LIN {X 0,Y 190.257,Z 771.261,A -85,B 0,C 180,E1 -26791.509,E2 -26791.509} C_VEL
LIN {X 0,Y 190.301,Z 771.078,A -85,B 0,C 180,E1 -26791.798,E2 -26791.798} C_VEL
LIN {X 0,Y 189.39,Z 772.436,A -85,B 0,C 180,E1 -26792.401,E2 -26792.401} C_VEL
LIN {X 0,Y 186.858,Z 776.269,A -85,B 0,C 180,E1 -26793.185,E2 -26793.185} C_VEL
LIN {X 0,Y 179.691,Z 786.165,A -85,B 0,C 180,E1 -26794.58,E2 -26794.58} C_VEL
LIN {X 0,Y 172.891,Z 794.099,A -85,B 0,C 180,E1 -26795.858,E2 -26795.858} C_VEL
LIN {X 0,Y 164.978,Z 801.951,A -85,B 0,C 180,E1 -26797.455,E2 -26797.455} C_VEL
LIN {X 0,Y 154.213,Z 810.811,A -85,B 0,C 180,E1 -26800.013,E2 -26800.013} C_VEL
LIN {X 0,Y 146.324,Z 816.184,A -85,B 0,C 180,E1 -26802.169,E2 -26802.169} C_VEL
LIN {X 0,Y 137.196,Z 821.36,A -85,B 0,C 180,E1 -26805.159,E2 -26805.159} C_VEL
LIN {X 0,Y 129.179,Z 825.032,A -85,B 0,C 180,E1 -26808.3,E2 -26808.3} C_VEL
LIN {X 0,Y 120.494,Z 828.105,A -85,B 0,C 180,E1 -26812.517,E2 -26812.517} C_VEL
LIN {X 0,Y 112.556,Z 829.932,A -85,B 0,C 180,E1 -26817.398,E2 -26817.398} C_VEL
LIN {X 0,Y 104.804,Z 830.561,A -85,B 0,C 180,E1 -26823.845,E2 -26823.845} C_VEL
LIN {X 0,Y 99.766,Z 830.01,A -85,B 0,C 180,E1 -26829.549,E2 -26829.549} C_VEL
LIN {X 0,Y 95.081,Z 828.076,A -85,B 0,C 180,E1 -26837.197,E2 -26837.197} C_VEL
LIN {X 0,Y 92.422,Z 825.28,A -85,B 0,C 180,E1 -26844.158,E2 -26844.158} C_VEL
LIN {X 0,Y 91.047,Z 820.547,A -85,B 0,C 180,E1 -26852.706,E2 -26852.706} C_VEL
LIN {X 0,Y 91.19,Z 815.515,A -85,B 0,C 180,E1 -26859.592,E2 -26859.592} C_VEL
LIN {X 0,Y 91.968,Z 810.446,A -85,B 0,C 180,E1 -26865.175,E2 -26865.175} C_VEL
LIN {X 0,Y 93.476,Z 803.521,A -85,B 0,C 180,E1 -26871.266,E2 -26871.266} C_VEL
LIN {X 0,Y 95.726,Z 795.077,A -85,B 0,C 180,E1 -26877.134,E2 -26877.134} C_VEL
LIN {X 0,Y 98.846,Z 784.708,A -85,B 0,C 180,E1 -26882.716,E2 -26882.716} C_VEL
LIN {X 0,Y 102.013,Z 773.87,A -85,B 0,C 180,E1 -26887.138,E2 -26887.138} C_VEL
LIN {X 0,Y 105.077,Z 762.843,A -85,B 0,C 180,E1 -26890.585,E2 -26890.585} C_VEL
LIN {X 0,Y 107.937,Z 750.627,A -85,B 0,C 180,E1 -26893.49,E2 -26893.49} C_VEL
LIN {X 0,Y 110.363,Z 737.817,A -85,B 0,C 180,E1 -26895.696,E2 -26895.696} C_VEL
LIN {X 0,Y 112.229,Z 724.1,A -85,B 0,C 180,E1 -26897.338,E2 -26897.338} C_VEL
LIN {X 0,Y 116.253,Z 682.181,A -85,B 0,C 180,E1 -26900.432,E2 -26900.432} C_VEL
LIN {X 0,Y 115.274,Z 679.01,A -85,B 0,C 180,E1 -26901.012,E2 -26901.012} C_VEL
LIN {X 0,Y 108.762,Z 662.742,A -85,B 0,C 180,E1 -26904.591,E2 -26904.591} C_VEL
LIN {X 0,Y 103.474,Z 650.911,A -85,B 0,C 180,E1 -26907.786,E2 -26907.786} C_VEL
LIN {X 0,Y 97.006,Z 638.252,A -85,B 0,C 180,E1 -26912.011,E2 -26912.011} C_VEL
LIN {X 0,Y 95.064,Z 635.94,A -85,B 0,C 180,E1 -26913.23,E2 -26913.23} C_VEL
LIN {X 0,Y 94.335,Z 633.735,A -85,B 0,C 180,E1 -26914.036,E2 -26914.036} C_VEL
LIN {X 0,Y 94.213,Z 633.749,A -85,B 0,C 180,E1 -26918.585,E2 -26918.585} C_VEL
LIN {X 0,Y 94.049,Z 633.77,A -85,B 0,C 180,E1 -26923.726,E2 -26923.726} C_VEL
LIN {X 0,Y 93.696,Z 633.798,A -85,B 0,C 180,E1 -26932.032,E2 -26932.032} C_VEL
LIN {X 0,Y 93.625,Z 633.822,A -85,B 0,C 180,E1 -26936.774,E2 -26936.774} C_VEL
LIN {X 0,Y 93.591,Z 633.786,A -85,B 0,C 180,E1 -26944.309,E2 -26944.309} C_VEL
LIN {X 0,Y 93.537,Z 633.831,A -85,B 0,C 180,E1 -26952.555,E2 -26952.555} C_VEL
LIN {X 0,Y 93.542,Z 633.801,A -85,B 0,C 180,E1 -26958.711,E2 -26958.711} C_VEL
LIN {X 0,Y 93.596,Z 633.788,A -85,B 0,C 180,E1 -26965.695,E2 -26965.695} C_VEL
LIN {X 0,Y 93.675,Z 633.815,A -85,B 0,C 180,E1 -26974.208,E2 -26974.208} C_VEL
LIN {X 0,Y 93.696,Z 633.798,A -85,B 0,C 180,E1 -26977.974,E2 -26977.974} C_VEL
LIN {X 0,Y 94.075,Z 633.734,A -85,B 0,C 180,E1 -26987.05,E2 -26987.05} C_VEL
LIN {X 0,Y 94.184,Z 633.749,A -85,B 0,C 180,E1 -26991.418,E2 -26991.418} C_VEL
LIN {X 0,Y 94.782,Z 633.646,A -85,B 0,C 180,E1 -27000.001,E2 -27000.001} C_VEL
LIN {X 0,Y 94.172,Z 633.755,A -85,B 0,C 180,E1 -27008.585,E2 -27008.585} C_VEL
LIN {X 0,Y 93.971,Z 633.763,A -85,B 0,C 180,E1 -27013.51,E2 -27013.51} C_VEL
LIN {X 0,Y 93.693,Z 633.817,A -85,B 0,C 180,E1 -27022.028,E2 -27022.028} C_VEL
LIN {X 0,Y 93.627,Z 633.827,A -85,B 0,C 180,E1 -27029.204,E2 -27029.204} C_VEL
LIN {X 0,Y 93.635,Z 633.826,A -85,B 0,C 180,E1 -27029.51,E2 -27029.51} C_VEL
LIN {X 0,Y 94.623,Z 636.565,A -85,B 0,C 180,E1 -27030.398,E2 -27030.398} C_VEL
LIN {X 0,Y 96.199,Z 638.846,A -85,B 0,C 180,E1 -27031.453,E2 -27031.453} C_VEL
LIN {X 0,Y 103.193,Z 651.438,A -85,B 0,C 180,E1 -27035.955,E2 -27035.955} C_VEL
LIN {X 0,Y 108.688,Z 666.292,A -85,B 0,C 180,E1 -27039.528,E2 -27039.528} C_VEL
LIN {X 0,Y 114.31,Z 684.536,A -85,B 0,C 180,E1 -27043.054,E2 -27043.054} C_VEL
LIN {X 0,Y 115.161,Z 702.412,A -85,B 0,C 180,E1 -27045.026,E2 -27045.026} C_VEL
LIN {X 0,Y 111.773,Z 738.131,A -85,B 0,C 180,E1 -27047.773,E2 -27047.773} C_VEL
LIN {X 0,Y 109.635,Z 752.163,A -85,B 0,C 180,E1 -27049.525,E2 -27049.525} C_VEL
LIN {X 0,Y 107.125,Z 764.111,A -85,B 0,C 180,E1 -27051.681,E2 -27051.681} C_VEL
LIN {X 0,Y 103.733,Z 777.276,A -85,B 0,C 180,E1 -27054.978,E2 -27054.978} C_VEL
LIN {X 0,Y 100.451,Z 788.747,A -85,B 0,C 180,E1 -27058.932,E2 -27058.932} C_VEL
LIN {X 0,Y 97.658,Z 798.326,A -85,B 0,C 180,E1 -27063.265,E2 -27063.265} C_VEL
LIN {X 0,Y 95.188,Z 807.085,A -85,B 0,C 180,E1 -27068.331,E2 -27068.331} C_VEL
LIN {X 0,Y 93.458,Z 814.321,A -85,B 0,C 180,E1 -27073.616,E2 -27073.616} C_VEL
LIN {X 0,Y 92.315,Z 821.391,A -85,B 0,C 180,E1 -27080.132,E2 -27080.132} C_VEL
LIN {X 0,Y 92.185,Z 826.13,A -85,B 0,C 180,E1 -27085.623,E2 -27085.623} C_VEL
LIN {X 0,Y 92.19,Z 829.203,A -85,B 0,C 180,E1 -27089.995,E2 -27089.995} C_VEL
LIN {X 0,Y 91.921,Z 832.559,A -85,B 0,C 180,E1 -27096.306,E2 -27096.306} C_VEL
LIN {X 0,Y 92.284,Z 835.092,A -85,B 0,C 180,E1 -27103.202,E2 -27103.202} C_VEL
LIN {X 0,Y 94.653,Z 837.065,A -85,B 0,C 180,E1 -27111.788,E2 -27111.788} C_VEL
LIN {X 0,Y 99.342,Z 837.643,A -85,B 0,C 180,E1 -27119.679,E2 -27119.679} C_VEL
LIN {X 0,Y 105.831,Z 836.874,A -85,B 0,C 180,E1 -27126.698,E2 -27126.698} C_VEL
LIN {X 0,Y 113.876,Z 834.76,A -85,B 0,C 180,E1 -27132.751,E2 -27132.751} C_VEL
LIN {X 0,Y 123.232,Z 831.198,A -85,B 0,C 180,E1 -27137.845,E2 -27137.845} C_VEL
LIN {X 0,Y 133.648,Z 826.087,A -85,B 0,C 180,E1 -27142.067,E2 -27142.067} C_VEL
LIN {X 0,Y 142.003,Z 821.149,A -85,B 0,C 180,E1 -27144.742,E2 -27144.742} C_VEL
LIN {X 0,Y 152.185,Z 813.997,A -85,B 0,C 180,E1 -27147.431,E2 -27147.431} C_VEL
LIN {X 0,Y 161.26,Z 806.403,A -85,B 0,C 180,E1 -27149.394,E2 -27149.394} C_VEL
LIN {X 0,Y 170.664,Z 797.142,A -85,B 0,C 180,E1 -27151.049,E2 -27151.049} C_VEL
LIN {X 0,Y 179.448,Z 786.784,A -85,B 0,C 180,E1 -27152.381,E2 -27152.381} C_VEL
LIN {X 0,Y 184.99,Z 779.053,A -85,B 0,C 180,E1 -27153.104,E2 -27153.104} C_VEL
LIN {X 0,Y 185.21,Z 778.645,A -85,B 0,C 180,E1 -27153.656,E2 -27153.656} C_VEL
LIN {X 0,Y 177.086,Z 789.352,A -85,B 0,C 180,E1 -27155.058,E2 -27155.058} C_VEL
LIN {X 0,Y 172.891,Z 794.099,A -85,B 0,C 180,E1 -27155.858,E2 -27155.858} C_VEL
LIN {X 0,Y 168.899,Z 798.22,A -85,B 0,C 180,E1 -27156.407,E2 -27156.407} C_VEL
LIN {X 0,Y 161.572,Z 804.876,A -85,B 0,C 180,E1 -27156.817,E2 -27156.817} C_VEL
LIN {X 0,Y 153.89,Z 810.838,A -85,B 0,C 180,E1 -27157.356,E2 -27157.356} C_VEL
LIN {X 0,Y 149.397,Z 813.899,A -85,B 0,C 180,E1 -27158.148,E2 -27158.148} C_VEL
LIN {X 0,Y 139.254,Z 819.917,A -85,B 0,C 180,E1 -27160.848,E2 -27160.848} C_VEL
LIN {X 0,Y 129.108,Z 824.664,A -85,B 0,C 180,E1 -27164.206,E2 -27164.206} C_VEL
LIN {X 0,Y 122.663,Z 827.054,A -85,B 0,C 180,E1 -27166.751,E2 -27166.751} C_VEL
LIN {X 0,Y 113.839,Z 829.524,A -85,B 0,C 180,E1 -27171.006,E2 -27171.006} C_VEL
LIN {X 0,Y 105.533,Z 830.874,A -85,B 0,C 180,E1 -27176.181,E2 -27176.181} C_VEL
LIN {X 0,Y 98.447,Z 831.013,A -85,B 0,C 180,E1 -27182.063,E2 -27182.063} C_VEL
LIN {X 0,Y 92.478,Z 829.966,A -85,B 0,C 180,E1 -27188.933,E2 -27188.933} C_VEL
LIN {X 0,Y 87.974,Z 827.723,A -85,B 0,C 180,E1 -27196.554,E2 -27196.554} C_VEL
LIN {X 0,Y 85.101,Z 824.276,A -85,B 0,C 180,E1 -27204.725,E2 -27204.725} C_VEL
LIN {X 0,Y 83.943,Z 819.532,A -85,B 0,C 180,E1 -27213.161,E2 -27213.161} C_VEL
LIN {X 0,Y 84.158,Z 814.597,A -85,B 0,C 180,E1 -27220.015,E2 -27220.015} C_VEL
LIN {X 0,Y 85.397,Z 807.511,A -85,B 0,C 180,E1 -27227.789,E2 -27227.789} C_VEL
LIN {X 0,Y 87.491,Z 799.088,A -85,B 0,C 180,E1 -27234.89,E2 -27234.89} C_VEL
LIN {X 0,Y 90.326,Z 789.576,A -85,B 0,C 180,E1 -27241.072,E2 -27241.072} C_VEL
LIN {X 0,Y 93.463,Z 779.613,A -85,B 0,C 180,E1 -27245.988,E2 -27245.988} C_VEL
LIN {X 0,Y 96.948,Z 767.721,A -85,B 0,C 180,E1 -27250.458,E2 -27250.458} C_VEL
LIN {X 0,Y 99.998,Z 756.271,A -85,B 0,C 180,E1 -27253.677,E2 -27253.677} C_VEL
LIN {X 0,Y 102.829,Z 743.465,A -85,B 0,C 180,E1 -27256.32,E2 -27256.32} C_VEL
LIN {X 0,Y 105.103,Z 729.84,A -85,B 0,C 180,E1 -27258.31,E2 -27258.31} C_VEL
LIN {X 0,Y 107.076,Z 711.899,A -85,B 0,C 180,E1 -27259.909,E2 -27259.909} C_VEL
LIN {X 0,Y 109.842,Z 683.218,A -85,B 0,C 180,E1 -27262.095,E2 -27262.095} C_VEL
LIN {X 0,Y 103.379,Z 666.533,A -85,B 0,C 180,E1 -27266.022,E2 -27266.022} C_VEL
LIN {X 0,Y 98.287,Z 654.89,A -85,B 0,C 180,E1 -27269.36,E2 -27269.36} C_VEL
LIN {X 0,Y 92.53,Z 643.401,A -85,B 0,C 180,E1 -27273.467,E2 -27273.467} C_VEL
LIN {X 0,Y 90.263,Z 640.187,A -85,B 0,C 180,E1 -27275.111,E2 -27275.111} C_VEL
LIN {X 0,Y 89.464,Z 638.976,A -85,B 0,C 180,E1 -27275.726,E2 -27275.726} C_VEL
LIN {X 0,Y 87.736,Z 636.65,A -85,B 0,C 180,E1 -27277.051,E2 -27277.051} C_VEL
LIN {X 0,Y 87.154,Z 634.627,A -85,B 0,C 180,E1 -27277.826,E2 -27277.826} C_VEL
LIN {X 0,Y 86.952,Z 634.654,A -85,B 0,C 180,E1 -27284.092,E2 -27284.092} C_VEL
LIN {X 0,Y 86.59,Z 634.695,A -85,B 0,C 180,E1 -27293.948,E2 -27293.948} C_VEL
LIN {X 0,Y 86.478,Z 634.702,A -85,B 0,C 180,E1 -27299.189,E2 -27299.189} C_VEL
LIN {X 0,Y 86.51,Z 634.671,A -85,B 0,C 180,E1 -27305.67,E2 -27305.67} C_VEL
LIN {X 0,Y 86.481,Z 634.71,A -85,B 0,C 180,E1 -27312.997,E2 -27312.997} C_VEL
LIN {X 0,Y 86.464,Z 634.672,A -85,B 0,C 180,E1 -27319.44,E2 -27319.44} C_VEL
LIN {X 0,Y 86.54,Z 634.661,A -85,B 0,C 180,E1 -27325.357,E2 -27325.357} C_VEL
LIN {X 0,Y 86.59,Z 634.699,A -85,B 0,C 180,E1 -27333.238,E2 -27333.238} C_VEL
LIN {X 0,Y 86.638,Z 634.648,A -85,B 0,C 180,E1 -27341.067,E2 -27341.067} C_VEL
LIN {X 0,Y 86.938,Z 634.611,A -85,B 0,C 180,E1 -27345.965,E2 -27345.965} C_VEL
LIN {X 0,Y 87.093,Z 634.629,A -85,B 0,C 180,E1 -27350.713,E2 -27350.713} C_VEL
LIN {X 0,Y 87.712,Z 634.525,A -85,B 0,C 180,E1 -27360.001,E2 -27360.001} C_VEL
LIN {X 0,Y 87.074,Z 634.639,A -85,B 0,C 180,E1 -27369.29,E2 -27369.29} C_VEL
LIN {X 0,Y 86.868,Z 634.644,A -85,B 0,C 180,E1 -27374.047,E2 -27374.047} C_VEL
LIN {X 0,Y 86.627,Z 634.693,A -85,B 0,C 180,E1 -27378.937,E2 -27378.937} C_VEL
LIN {X 0,Y 86.629,Z 634.683,A -85,B 0,C 180,E1 -27385.699,E2 -27385.699} C_VEL
LIN {X 0,Y 87.657,Z 637.659,A -85,B 0,C 180,E1 -27386.827,E2 -27386.827} C_VEL
LIN {X 0,Y 89.274,Z 639.751,A -85,B 0,C 180,E1 -27388.058,E2 -27388.058} C_VEL
LIN {X 0,Y 95.254,Z 650.213,A -85,B 0,C 180,E1 -27392.495,E2 -27392.495} C_VEL
LIN {X 0,Y 98.46,Z 656.546,A -85,B 0,C 180,E1 -27394.668,E2 -27394.668} C_VEL
LIN {X 0,Y 104.026,Z 672.659,A -85,B 0,C 180,E1 -27398.678,E2 -27398.678} C_VEL
LIN {X 0,Y 108.21,Z 687.138,A -85,B 0,C 180,E1 -27401.583,E2 -27401.583} C_VEL
LIN {X 0,Y 108.806,Z 702.893,A -85,B 0,C 180,E1 -27403.389,E2 -27403.389} C_VEL
LIN {X 0,Y 105.359,Z 737.654,A -85,B 0,C 180,E1 -27406.201,E2 -27406.201} C_VEL
LIN {X 0,Y 103.128,Z 751.621,A -85,B 0,C 180,E1 -27408.028,E2 -27408.028} C_VEL
LIN {X 0,Y 100.378,Z 764.08,A -85,B 0,C 180,E1 -27410.41,E2 -27410.41} C_VEL
LIN {X 0,Y 97.072,Z 776.396,A -85,B 0,C 180,E1 -27413.681,E2 -27413.681} C_VEL
LIN {X 0,Y 93.764,Z 787.607,A -85,B 0,C 180,E1 -27417.715,E2 -27417.715} C_VEL
LIN {X 0,Y 90.803,Z 797.289,A -85,B 0,C 180,E1 -27422.324,E2 -27422.324} C_VEL
LIN {X 0,Y 88.22,Z 806.145,A -85,B 0,C 180,E1 -27427.76,E2 -27427.76} C_VEL
LIN {X 0,Y 86.147,Z 814.79,A -85,B 0,C 180,E1 -27434.62,E2 -27434.62} C_VEL
LIN {X 0,Y 85.214,Z 821.7,A -85,B 0,C 180,E1 -27441.773,E2 -27441.773} C_VEL
LIN {X 0,Y 85.191,Z 826.219,A -85,B 0,C 180,E1 -27447.631,E2 -27447.631} C_VEL
LIN {X 0,Y 85.153,Z 829.094,A -85,B 0,C 180,E1 -27452.36,E2 -27452.36} C_VEL
LIN {X 0,Y 84.943,Z 832.374,A -85,B 0,C 180,E1 -27459.52,E2 -27459.52} C_VEL
LIN {X 0,Y 86.475,Z 835.317,A -85,B 0,C 180,E1 -27468.965,E2 -27468.965} C_VEL
LIN {X 0,Y 90.35,Z 836.847,A -85,B 0,C 180,E1 -27477.816,E2 -27477.816} C_VEL
LIN {X 0,Y 96.496,Z 837.06,A -85,B 0,C 180,E1 -27485.632,E2 -27485.632} C_VEL
LIN {X 0,Y 104.304,Z 835.891,A -85,B 0,C 180,E1 -27492.355,E2 -27492.355} C_VEL
LIN {X 0,Y 113.522,Z 833.378,A -85,B 0,C 180,E1 -27497.973,E2 -27497.973} C_VEL
LIN {X 0,Y 121.231,Z 830.566,A -85,B 0,C 180,E1 -27501.495,E2 -27501.495} C_VEL
LIN {X 0,Y 132.291,Z 825.471,A -85,B 0,C 180,E1 -27505.424,E2 -27505.424} C_VEL
LIN {X 0,Y 141.025,Z 820.498,A -85,B 0,C 180,E1 -27507.902,E2 -27507.902} C_VEL
LIN {X 0,Y 151.627,Z 813.379,A -85,B 0,C 180,E1 -27510.345,E2 -27510.345} C_VEL
LIN {X 0,Y 161.018,Z 805.796,A -85,B 0,C 180,E1 -27512.105,E2 -27512.105} C_VEL
LIN {X 0,Y 167.484,Z 799.75,A -85,B 0,C 180,E1 -27513.122,E2 -27513.122} C_VEL
LIN {X 0,Y 169.396,Z 797.758,A -85,B 0,C 180,E1 -27513.97,E2 -27513.97} C_VEL
LIN {X 0,Y 160.59,Z 805.702,A -85,B 0,C 180,E1 -27515.652,E2 -27515.652} C_VEL
LIN {X 0,Y 150.031,Z 813.478,A -85,B 0,C 180,E1 -27517.991,E2 -27517.991} C_VEL
LIN {X 0,Y 149.397,Z 813.899,A -85,B 0,C 180,E1 -27518.148,E2 -27518.148} C_VEL
LIN {X 0,Y 144.757,Z 816.802,A -85,B 0,C 180,E1 -27519.036,E2 -27519.036} C_VEL
LIN {X 0,Y 136.239,Z 821.334,A -85,B 0,C 180,E1 -27520.012,E2 -27520.012} C_VEL
LIN {X 0,Y 127.551,Z 825.143,A -85,B 0,C 180,E1 -27521.2,E2 -27521.2} C_VEL
LIN {X 0,Y 122.718,Z 826.849,A -85,B 0,C 180,E1 -27522.485,E2 -27522.485} C_VEL
LIN {X 0,Y 114.479,Z 829.304,A -85,B 0,C 180,E1 -27525.784,E2 -27525.784} C_VEL
LIN {X 0,Y 107.282,Z 830.741,A -85,B 0,C 180,E1 -27529.285,E2 -27529.285} C_VEL
LIN {X 0,Y 98.829,Z 831.572,A -85,B 0,C 180,E1 -27534.558,E2 -27534.558} C_VEL
LIN {X 0,Y 91.366,Z 831.247,A -85,B 0,C 180,E1 -27540.858,E2 -27540.858} C_VEL
LIN {X 0,Y 85.202,Z 829.729,A -85,B 0,C 180,E1 -27548.214,E2 -27548.214} C_VEL
LIN {X 0,Y 80.612,Z 826.993,A -85,B 0,C 180,E1 -27556.482,E2 -27556.482} C_VEL
LIN {X 0,Y 77.813,Z 823.015,A -85,B 0,C 180,E1 -27565.434,E2 -27565.434} C_VEL
LIN {X 0,Y 76.866,Z 817.762,A -85,B 0,C 180,E1 -27574.636,E2 -27574.636} C_VEL
LIN {X 0,Y 77.27,Z 812.753,A -85,B 0,C 180,E1 -27581.579,E2 -27581.579} C_VEL
LIN {X 0,Y 78.524,Z 806.204,A -85,B 0,C 180,E1 -27588.885,E2 -27588.885} C_VEL
LIN {X 0,Y 80.91,Z 797.234,A -85,B 0,C 180,E1 -27596.678,E2 -27596.678} C_VEL
LIN {X 0,Y 84.32,Z 786.507,A -85,B 0,C 180,E1 -27603.637,E2 -27603.637} C_VEL
LIN {X 0,Y 87.783,Z 775.869,A -85,B 0,C 180,E1 -27608.795,E2 -27608.795} C_VEL
LIN {X 0,Y 91.421,Z 763.754,A -85,B 0,C 180,E1 -27613.167,E2 -27613.167} C_VEL
LIN {X 0,Y 94.498,Z 752.043,A -85,B 0,C 180,E1 -27616.297,E2 -27616.297} C_VEL
LIN {X 0,Y 97.388,Z 738.237,A -85,B 0,C 180,E1 -27618.911,E2 -27618.911} C_VEL
LIN {X 0,Y 99.344,Z 725.28,A -85,B 0,C 180,E1 -27620.602,E2 -27620.602} C_VEL
LIN {X 0,Y 103.501,Z 684.743,A -85,B 0,C 180,E1 -27623.911,E2 -27623.911} C_VEL
LIN {X 0,Y 97.838,Z 669.858,A -85,B 0,C 180,E1 -27627.699,E2 -27627.699} C_VEL
LIN {X 0,Y 93.131,Z 658.831,A -85,B 0,C 180,E1 -27631.087,E2 -27631.087} C_VEL
LIN {X 0,Y 87.987,Z 648.291,A -85,B 0,C 180,E1 -27635.173,E2 -27635.173} C_VEL
LIN {X 0,Y 84.861,Z 643.815,A -85,B 0,C 180,E1 -27637.652,E2 -27637.652} C_VEL
LIN {X 0,Y 82.422,Z 639.977,A -85,B 0,C 180,E1 -27639.824,E2 -27639.824} C_VEL
LIN {X 0,Y 80.655,Z 637.846,A -85,B 0,C 180,E1 -27641.419,E2 -27641.419} C_VEL
LIN {X 0,Y 79.921,Z 635.526,A -85,B 0,C 180,E1 -27642.481,E2 -27642.481} C_VEL
LIN {X 0,Y 79.516,Z 635.555,A -85,B 0,C 180,E1 -27650.71,E2 -27650.71} C_VEL
LIN {X 0,Y 79.485,Z 635.58,A -85,B 0,C 180,E1 -27657.849,E2 -27657.849} C_VEL
LIN {X 0,Y 79.381,Z 635.559,A -85,B 0,C 180,E1 -27662.094,E2 -27662.094} C_VEL
LIN {X 0,Y 79.369,Z 635.58,A -85,B 0,C 180,E1 -27668.311,E2 -27668.311} C_VEL
LIN {X 0,Y 79.39,Z 635.586,A -85,B 0,C 180,E1 -27675.096,E2 -27675.096} C_VEL
LIN {X 0,Y 79.393,Z 635.536,A -85,B 0,C 180,E1 -27682.824,E2 -27682.824} C_VEL
LIN {X 0,Y 79.385,Z 635.575,A -85,B 0,C 180,E1 -27687.915,E2 -27687.915} C_VEL
LIN {X 0,Y 79.531,Z 635.578,A -85,B 0,C 180,E1 -27693.779,E2 -27693.779} C_VEL
LIN {X 0,Y 79.511,Z 635.549,A -85,B 0,C 180,E1 -27699.296,E2 -27699.296} C_VEL
LIN {X 0,Y 79.832,Z 635.491,A -85,B 0,C 180,E1 -27705.575,E2 -27705.575} C_VEL
LIN {X 0,Y 79.976,Z 635.511,A -85,B 0,C 180,E1 -27709.878,E2 -27709.878} C_VEL
LIN {X 0,Y 80.641,Z 635.404,A -85,B 0,C 180,E1 -27720.001,E2 -27720.001} C_VEL
LIN {X 0,Y 79.951,Z 635.526,A -85,B 0,C 180,E1 -27730.126,E2 -27730.126} C_VEL
LIN {X 0,Y 79.7,Z 635.535,A -85,B 0,C 180,E1 -27735.341,E2 -27735.341} C_VEL
LIN {X 0,Y 79.508,Z 635.586,A -85,B 0,C 180,E1 -27741.046,E2 -27741.046} C_VEL
LIN {X 0,Y 80.462,Z 638.379,A -85,B 0,C 180,E1 -27742.298,E2 -27742.298} C_VEL
LIN {X 0,Y 82.444,Z 640.682,A -85,B 0,C 180,E1 -27744.054,E2 -27744.054} C_VEL
LIN {X 0,Y 84.504,Z 644.136,A -85,B 0,C 180,E1 -27745.936,E2 -27745.936} C_VEL
LIN {X 0,Y 88.954,Z 651.914,A -85,B 0,C 180,E1 -27749.662,E2 -27749.662} C_VEL
LIN {X 0,Y 93.093,Z 659.974,A -85,B 0,C 180,E1 -27752.802,E2 -27752.802} C_VEL
LIN {X 0,Y 98.329,Z 675.548,A -85,B 0,C 180,E1 -27756.93,E2 -27756.93} C_VEL
LIN {X 0,Y 102.085,Z 689.101,A -85,B 0,C 180,E1 -27759.876,E2 -27759.876} C_VEL
LIN {X 0,Y 102.526,Z 703.086,A -85,B 0,C 180,E1 -27761.586,E2 -27761.586} C_VEL
LIN {X 0,Y 98.903,Z 737.844,A -85,B 0,C 180,E1 -27764.551,E2 -27764.551} C_VEL
LIN {X 0,Y 96.715,Z 750.887,A -85,B 0,C 180,E1 -27766.34,E2 -27766.34} C_VEL
LIN {X 0,Y 93.883,Z 763.305,A -85,B 0,C 180,E1 -27768.803,E2 -27768.803} C_VEL
LIN {X 0,Y 90.418,Z 775.691,A -85,B 0,C 180,E1 -27772.252,E2 -27772.252} C_VEL
LIN {X 0,Y 87.128,Z 786.446,A -85,B 0,C 180,E1 -27776.314,E2 -27776.314} C_VEL
LIN {X 0,Y 83.991,Z 796.258,A -85,B 0,C 180,E1 -27781.235,E2 -27781.235} C_VEL
LIN {X 0,Y 81.262,Z 805.169,A -85,B 0,C 180,E1 -27787.09,E2 -27787.09} C_VEL
LIN {X 0,Y 79.113,Z 813.861,A -85,B 0,C 180,E1 -27794.538,E2 -27794.538} C_VEL
LIN {X 0,Y 78.268,Z 819.777,A -85,B 0,C 180,E1 -27801.021,E2 -27801.021} C_VEL
LIN {X 0,Y 78.216,Z 824.532,A -85,B 0,C 180,E1 -27807.419,E2 -27807.419} C_VEL
LIN {X 0,Y 78.216,Z 827.636,A -85,B 0,C 180,E1 -27812.569,E2 -27812.569} C_VEL
LIN {X 0,Y 78.053,Z 831.117,A -85,B 0,C 180,E1 -27820.369,E2 -27820.369} C_VEL
LIN {X 0,Y 79.815,Z 834.326,A -85,B 0,C 180,E1 -27830.617,E2 -27830.617} C_VEL
LIN {X 0,Y 84.142,Z 836.113,A -85,B 0,C 180,E1 -27840.07,E2 -27840.07} C_VEL
LIN {X 0,Y 90.814,Z 836.584,A -85,B 0,C 180,E1 -27848.245,E2 -27848.245} C_VEL
LIN {X 0,Y 99.165,Z 835.742,A -85,B 0,C 180,E1 -27855.124,E2 -27855.124} C_VEL
LIN {X 0,Y 108.904,Z 833.581,A -85,B 0,C 180,E1 -27860.745,E2 -27860.745} C_VEL
LIN {X 0,Y 114.204,Z 831.967,A -85,B 0,C 180,E1 -27863.124,E2 -27863.124} C_VEL
LIN {X 0,Y 125.472,Z 827.624,A -85,B 0,C 180,E1 -27867.153,E2 -27867.153} C_VEL
LIN {X 0,Y 137.437,Z 821.736,A -85,B 0,C 180,E1 -27870.372,E2 -27870.372} C_VEL
LIN {X 0,Y 148.303,Z 815.015,A -85,B 0,C 180,E1 -27872.684,E2 -27872.684} C_VEL
LIN {X 0,Y 151.71,Z 812.646,A -85,B 0,C 180,E1 -27873.312,E2 -27873.312} C_VEL
LIN {X 0,Y 153.789,Z 811.02,A -85,B 0,C 180,E1 -27874.211,E2 -27874.211} C_VEL
LIN {X 0,Y 144.85,Z 816.764,A -85,B 0,C 180,E1 -27876.128,E2 -27876.128} C_VEL
LIN {X 0,Y 134.892,Z 821.992,A -85,B 0,C 180,E1 -27878.61,E2 -27878.61} C_VEL
LIN {X 0,Y 126.124,Z 825.668,A -85,B 0,C 180,E1 -27881.303,E2 -27881.303} C_VEL
LIN {X 0,Y 122.718,Z 826.849,A -85,B 0,C 180,E1 -27882.485,E2 -27882.485} C_VEL
LIN {X 0,Y 117.866,Z 828.409,A -85,B 0,C 180,E1 -27883.923,E2 -27883.923} C_VEL
LIN {X 0,Y 108.967,Z 830.518,A -85,B 0,C 180,E1 -27885.871,E2 -27885.871} C_VEL
LIN {X 0,Y 100.179,Z 831.798,A -85,B 0,C 180,E1 -27888.234,E2 -27888.234} C_VEL
LIN {X 0,Y 95.623,Z 832.034,A -85,B 0,C 180,E1 -27890.399,E2 -27890.399} C_VEL
LIN {X 0,Y 88.689,Z 831.868,A -85,B 0,C 180,E1 -27895.454,E2 -27895.454} C_VEL
LIN {X 0,Y 83.805,Z 831.164,A -85,B 0,C 180,E1 -27899.999,E2 -27899.999} C_VEL
LIN {X 0,Y 77.942,Z 829.266,A -85,B 0,C 180,E1 -27907.361,E2 -27907.361} C_VEL
LIN {X 0,Y 73.086,Z 825.893,A -85,B 0,C 180,E1 -27916.766,E2 -27916.766} C_VEL
LIN {X 0,Y 70.266,Z 820.665,A -85,B 0,C 180,E1 -27927.957,E2 -27927.957} C_VEL
LIN {X 0,Y 69.872,Z 815.241,A -85,B 0,C 180,E1 -27937.12,E2 -27937.12} C_VEL
LIN {X 0,Y 70.815,Z 808.603,A -85,B 0,C 180,E1 -27946.005,E2 -27946.005} C_VEL
LIN {X 0,Y 72.417,Z 801.973,A -85,B 0,C 180,E1 -27953.038,E2 -27953.038} C_VEL
LIN {X 0,Y 75.148,Z 792.909,A -85,B 0,C 180,E1 -27960.492,E2 -27960.492} C_VEL
LIN {X 0,Y 78.482,Z 783.112,A -85,B 0,C 180,E1 -27966.617,E2 -27966.617} C_VEL
LIN {X 0,Y 81.681,Z 773.603,A -85,B 0,C 180,E1 -27971.165,E2 -27971.165} C_VEL
LIN {X 0,Y 85.317,Z 761.99,A -85,B 0,C 180,E1 -27975.363,E2 -27975.363} C_VEL
LIN {X 0,Y 88.684,Z 749.213,A -85,B 0,C 180,E1 -27978.719,E2 -27978.719} C_VEL
LIN {X 0,Y 91.427,Z 736.122,A -85,B 0,C 180,E1 -27981.161,E2 -27981.161} C_VEL
LIN {X 0,Y 93.491,Z 721.573,A -85,B 0,C 180,E1 -27982.939,E2 -27982.939} C_VEL
LIN {X 0,Y 97.333,Z 686.542,A -85,B 0,C 180,E1 -27985.864,E2 -27985.864} C_VEL
LIN {X 0,Y 91.872,Z 672.015,A -85,B 0,C 180,E1 -27989.893,E2 -27989.893} C_VEL
LIN {X 0,Y 87.991,Z 662.65,A -85,B 0,C 180,E1 -27993.073,E2 -27993.073} C_VEL
LIN {X 0,Y 83.41,Z 653.017,A -85,B 0,C 180,E1 -27997.066,E2 -27997.066} C_VEL
LIN {X 0,Y 78.246,Z 645.162,A -85,B 0,C 180,E1 -28001.881,E2 -28001.881} C_VEL
LIN {X 0,Y 76.263,Z 642.137,A -85,B 0,C 180,E1 -28004.024,E2 -28004.024} C_VEL
LIN {X 0,Y 75.71,Z 641.334,A -85,B 0,C 180,E1 -28004.637,E2 -28004.637} C_VEL
LIN {X 0,Y 73.425,Z 639.042,A -85,B 0,C 180,E1 -28007.12,E2 -28007.12} C_VEL
LIN {X 0,Y 72.482,Z 636.431,A -85,B 0,C 180,E1 -28008.629,E2 -28008.629} C_VEL
LIN {X 0,Y 72.397,Z 636.453,A -85,B 0,C 180,E1 -28012.855,E2 -28012.855} C_VEL
LIN {X 0,Y 72.38,Z 636.455,A -85,B 0,C 180,E1 -28019.088,E2 -28019.088} C_VEL
LIN {X 0,Y 72.297,Z 636.438,A -85,B 0,C 180,E1 -28025.687,E2 -28025.687} C_VEL
LIN {X 0,Y 72.25,Z 636.483,A -85,B 0,C 180,E1 -28032.923,E2 -28032.923} C_VEL
LIN {X 0,Y 72.3,Z 636.42,A -85,B 0,C 180,E1 -28041.055,E2 -28041.055} C_VEL
LIN {X 0,Y 72.301,Z 636.422,A -85,B 0,C 180,E1 -28044.323,E2 -28044.323} C_VEL
LIN {X 0,Y 72.381,Z 636.465,A -85,B 0,C 180,E1 -28050.956,E2 -28050.956} C_VEL
LIN {X 0,Y 72.396,Z 636.453,A -85,B 0,C 180,E1 -28057.151,E2 -28057.151} C_VEL
LIN {X 0,Y 72.727,Z 636.371,A -85,B 0,C 180,E1 -28065.117,E2 -28065.117} C_VEL
LIN {X 0,Y 72.866,Z 636.387,A -85,B 0,C 180,E1 -28068.879,E2 -28068.879} C_VEL
LIN {X 0,Y 73.568,Z 636.284,A -85,B 0,C 180,E1 -28080.001,E2 -28080.001} C_VEL
LIN {X 0,Y 72.836,Z 636.408,A -85,B 0,C 180,E1 -28091.128,E2 -28091.128} C_VEL
LIN {X 0,Y 72.657,Z 636.411,A -85,B 0,C 180,E1 -28095.24,E2 -28095.24} C_VEL
LIN {X 0,Y 73.572,Z 639.345,A -85,B 0,C 180,E1 -28096.832,E2 -28096.832} C_VEL
LIN {X 0,Y 75.625,Z 641.738,A -85,B 0,C 180,E1 -28099.158,E2 -28099.158} C_VEL
LIN {X 0,Y 77.626,Z 645.08,A -85,B 0,C 180,E1 -28101.407,E2 -28101.407} C_VEL
LIN {X 0,Y 80.948,Z 650.397,A -85,B 0,C 180,E1 -28104.698,E2 -28104.698} C_VEL
LIN {X 0,Y 85.717,Z 659.138,A -85,B 0,C 180,E1 -28108.965,E2 -28108.965} C_VEL
LIN {X 0,Y 88.26,Z 664.667,A -85,B 0,C 180,E1 -28111.137,E2 -28111.137} C_VEL
LIN {X 0,Y 92.625,Z 678.381,A -85,B 0,C 180,E1 -28115.017,E2 -28115.017} C_VEL
LIN {X 0,Y 96.044,Z 690.842,A -85,B 0,C 180,E1 -28117.93,E2 -28117.93} C_VEL
LIN {X 0,Y 96.354,Z 703.322,A -85,B 0,C 180,E1 -28119.57,E2 -28119.57} C_VEL
LIN {X 0,Y 92.569,Z 737.82,A -85,B 0,C 180,E1 -28122.647,E2 -28122.647} C_VEL
LIN {X 0,Y 90.143,Z 751.486,A -85,B 0,C 180,E1 -28124.651,E2 -28124.651} C_VEL
LIN {X 0,Y 86.952,Z 764.345,A -85,B 0,C 180,E1 -28127.453,E2 -28127.453} C_VEL
LIN {X 0,Y 83.136,Z 777.187,A -85,B 0,C 180,E1 -28131.425,E2 -28131.425} C_VEL
LIN {X 0,Y 79.378,Z 788.599,A -85,B 0,C 180,E1 -28136.396,E2 -28136.396} C_VEL
LIN {X 0,Y 75.984,Z 798.88,A -85,B 0,C 180,E1 -28142.447,E2 -28142.447} C_VEL
LIN {X 0,Y 73.083,Z 808.714,A -85,B 0,C 180,E1 -28150.325,E2 -28150.325} C_VEL
LIN {X 0,Y 71.465,Z 816.575,A -85,B 0,C 180,E1 -28158.651,E2 -28158.651} C_VEL
LIN {X 0,Y 71.237,Z 822.829,A -85,B 0,C 180,E1 -28167.166,E2 -28167.166} C_VEL
LIN {X 0,Y 71.313,Z 826.081,A -85,B 0,C 180,E1 -28172.818,E2 -28172.818} C_VEL
LIN {X 0,Y 71.201,Z 829.757,A -85,B 0,C 180,E1 -28181.379,E2 -28181.379} C_VEL
LIN {X 0,Y 73.265,Z 833.226,A -85,B 0,C 180,E1 -28192.557,E2 -28192.557} C_VEL
LIN {X 0,Y 78.092,Z 835.306,A -85,B 0,C 180,E1 -28202.675,E2 -28202.675} C_VEL
LIN {X 0,Y 85.347,Z 836.09,A -85,B 0,C 180,E1 -28211.199,E2 -28211.199} C_VEL
LIN {X 0,Y 94.282,Z 835.529,A -85,B 0,C 180,E1 -28218.188,E2 -28218.188} C_VEL
LIN {X 0,Y 104.568,Z 833.672,A -85,B 0,C 180,E1 -28223.75,E2 -28223.75} C_VEL
LIN {X 0,Y 110.106,Z 832.238,A -85,B 0,C 180,E1 -28226.069,E2 -28226.069} C_VEL
LIN {X 0,Y 121.792,Z 828.343,A -85,B 0,C 180,E1 -28229.941,E2 -28229.941} C_VEL
LIN {X 0,Y 130.985,Z 824.366,A -85,B 0,C 180,E1 -28232.281,E2 -28232.281} C_VEL
LIN {X 0,Y 136.102,Z 821.806,A -85,B 0,C 180,E1 -28233.4,E2 -28233.4} C_VEL
LIN {X 0,Y 138.341,Z 820.537,A -85,B 0,C 180,E1 -28234.407,E2 -28234.407} C_VEL
LIN {X 0,Y 127.066,Z 825.457,A -85,B 0,C 180,E1 -28237.221,E2 -28237.221} C_VEL
LIN {X 0,Y 118.861,Z 828.145,A -85,B 0,C 180,E1 -28239.747,E2 -28239.747} C_VEL
LIN {X 0,Y 110.284,Z 830.307,A -85,B 0,C 180,E1 -28242.906,E2 -28242.906} C_VEL
LIN {X 0,Y 99.959,Z 831.845,A -85,B 0,C 180,E1 -28247.823,E2 -28247.823} C_VEL
LIN {X 0,Y 95.623,Z 832.034,A -85,B 0,C 180,E1 -28250.399,E2 -28250.399} C_VEL
LIN {X 0,Y 91.202,Z 832.119,A -85,B 0,C 180,E1 -28252.803,E2 -28252.803} C_VEL
LIN {X 0,Y 83.038,Z 831.623,A -85,B 0,C 180,E1 -28256.489,E2 -28256.489} C_VEL
LIN {X 0,Y 75.348,Z 830.339,A -85,B 0,C 180,E1 -28260.927,E2 -28260.927} C_VEL
LIN {X 0,Y 71.855,Z 829.109,A -85,B 0,C 180,E1 -28264.541,E2 -28264.541} C_VEL
LIN {X 0,Y 67.61,Z 826.541,A -85,B 0,C 180,E1 -28271.998,E2 -28271.998} C_VEL
LIN {X 0,Y 64.086,Z 822.091,A -85,B 0,C 180,E1 -28282.57,E2 -28282.57} C_VEL
LIN {X 0,Y 62.807,Z 816.166,A -85,B 0,C 180,E1 -28294.02,E2 -28294.02} C_VEL
LIN {X 0,Y 63.38,Z 809.883,A -85,B 0,C 180,E1 -28303.64,E2 -28303.64} C_VEL
LIN {X 0,Y 64.903,Z 803.247,A -85,B 0,C 180,E1 -28311.726,E2 -28311.726} C_VEL
LIN {X 0,Y 67.387,Z 795.01,A -85,B 0,C 180,E1 -28319.63,E2 -28319.63} C_VEL
LIN {X 0,Y 70.764,Z 785.415,A -85,B 0,C 180,E1 -28326.6,E2 -28326.6} C_VEL
LIN {X 0,Y 74.453,Z 775.104,A -85,B 0,C 180,E1 -28332.178,E2 -28332.178} C_VEL
LIN {X 0,Y 78.134,Z 763.837,A -85,B 0,C 180,E1 -28336.704,E2 -28336.704} C_VEL
LIN {X 0,Y 81.465,Z 752.367,A -85,B 0,C 180,E1 -28340.07,E2 -28340.07} C_VEL
LIN {X 0,Y 84.695,Z 738.517,A -85,B 0,C 180,E1 -28342.931,E2 -28342.931} C_VEL
LIN {X 0,Y 86.933,Z 724.883,A -85,B 0,C 180,E1 -28344.814,E2 -28344.814} C_VEL
LIN {X 0,Y 91.106,Z 688.006,A -85,B 0,C 180,E1 -28348.091,E2 -28348.091} C_VEL
LIN {X 0,Y 85.617,Z 672.973,A -85,B 0,C 180,E1 -28352.798,E2 -28352.798} C_VEL
LIN {X 0,Y 81.875,Z 664.115,A -85,B 0,C 180,E1 -28356.21,E2 -28356.21} C_VEL
LIN {X 0,Y 78.867,Z 657.622,A -85,B 0,C 180,E1 -28359.208,E2 -28359.208} C_VEL
LIN {X 0,Y 74.21,Z 650.274,A -85,B 0,C 180,E1 -28364.134,E2 -28364.134} C_VEL
LIN {X 0,Y 72.005,Z 646.996,A -85,B 0,C 180,E1 -28366.744,E2 -28366.744} C_VEL
LIN {X 0,Y 69.701,Z 644.182,A -85,B 0,C 180,E1 -28369.646,E2 -28369.646} C_VEL
LIN {X 0,Y 68.89,Z 642.6,A -85,B 0,C 180,E1 -28370.905,E2 -28370.905} C_VEL
LIN {X 0,Y 66.34,Z 640.283,A -85,B 0,C 180,E1 -28374.606,E2 -28374.606} C_VEL
LIN {X 0,Y 65.385,Z 638.059,A -85,B 0,C 180,E1 -28376.54,E2 -28376.54} C_VEL
LIN {X 0,Y 65.251,Z 637.355,A -85,B 0,C 180,E1 -28377.06,E2 -28377.06} C_VEL
LIN {X 0,Y 65.199,Z 637.32,A -85,B 0,C 180,E1 -28382.621,E2 -28382.621} C_VEL
LIN {X 0,Y 65.186,Z 637.36,A -85,B 0,C 180,E1 -28391.002,E2 -28391.002} C_VEL
LIN {X 0,Y 65.207,Z 637.309,A -85,B 0,C 180,E1 -28399.709,E2 -28399.709} C_VEL
LIN {X 0,Y 65.26,Z 637.343,A -85,B 0,C 180,E1 -28409.502,E2 -28409.502} C_VEL
LIN {X 0,Y 65.243,Z 637.357,A -85,B 0,C 180,E1 -28414.477,E2 -28414.477} C_VEL
LIN {X 0,Y 65.631,Z 637.251,A -85,B 0,C 180,E1 -28424.551,E2 -28424.551} C_VEL
LIN {X 0,Y 65.762,Z 637.255,A -85,B 0,C 180,E1 -28427.659,E2 -28427.659} C_VEL
LIN {X 0,Y 65.923,Z 637.272,A -85,B 0,C 180,E1 -28433.881,E2 -28433.881} C_VEL
LIN {X 0,Y 66.466,Z 637.167,A -85,B 0,C 180,E1 -28440.001,E2 -28440.001} C_VEL
LIN {X 0,Y 65.849,Z 637.303,A -85,B 0,C 180,E1 -28447.668,E2 -28447.668} C_VEL
LIN {X 0,Y 66.559,Z 639.712,A -85,B 0,C 180,E1 -28449.306,E2 -28449.306} C_VEL
LIN {X 0,Y 68.726,Z 642.241,A -85,B 0,C 180,E1 -28452.575,E2 -28452.575} C_VEL
LIN {X 0,Y 71.132,Z 646.347,A -85,B 0,C 180,E1 -28456.031,E2 -28456.031} C_VEL
LIN {X 0,Y 72.308,Z 648.068,A -85,B 0,C 180,E1 -28457.5,E2 -28457.5} C_VEL
LIN {X 0,Y 76.308,Z 654.493,A -85,B 0,C 180,E1 -28462.151,E2 -28462.151} C_VEL
LIN {X 0,Y 81.153,Z 663.841,A -85,B 0,C 180,E1 -28467.044,E2 -28467.044} C_VEL
LIN {X 0,Y 83.274,Z 668.635,A -85,B 0,C 180,E1 -28469.031,E2 -28469.031} C_VEL
LIN {X 0,Y 87.191,Z 681.824,A -85,B 0,C 180,E1 -28473.057,E2 -28473.057} C_VEL
LIN {X 0,Y 90.036,Z 692.787,A -85,B 0,C 180,E1 -28475.837,E2 -28475.837} C_VEL
LIN {X 0,Y 90.145,Z 704.351,A -85,B 0,C 180,E1 -28477.408,E2 -28477.408} C_VEL
LIN {X 0,Y 86.341,Z 737.177,A -85,B 0,C 180,E1 -28480.482,E2 -28480.482} C_VEL
LIN {X 0,Y 83.854,Z 750.663,A -85,B 0,C 180,E1 -28482.544,E2 -28482.544} C_VEL
LIN {X 0,Y 80.793,Z 762.635,A -85,B 0,C 180,E1 -28485.204,E2 -28485.204} C_VEL
LIN {X 0,Y 76.825,Z 775.541,A -85,B 0,C 180,E1 -28489.316,E2 -28489.316} C_VEL
LIN {X 0,Y 73.194,Z 786.057,A -85,B 0,C 180,E1 -28493.969,E2 -28493.969} C_VEL
LIN {X 0,Y 69.813,Z 795.723,A -85,B 0,C 180,E1 -28499.772,E2 -28499.772} C_VEL
LIN {X 0,Y 66.975,Z 804.575,A -85,B 0,C 180,E1 -28506.82,E2 -28506.82} C_VEL
LIN {X 0,Y 64.83,Z 813.162,A -85,B 0,C 180,E1 -28515.875,E2 -28515.875} C_VEL
LIN {X 0,Y 64.243,Z 819.959,A -85,B 0,C 180,E1 -28525.287,E2 -28525.287} C_VEL
LIN {X 0,Y 64.4,Z 824.408,A -85,B 0,C 180,E1 -28533.121,E2 -28533.121} C_VEL
LIN {X 0,Y 64.372,Z 828.307,A -85,B 0,C 180,E1 -28542.605,E2 -28542.605} C_VEL
LIN {X 0,Y 66.831,Z 832.087,A -85,B 0,C 180,E1 -28554.868,E2 -28554.868} C_VEL
LIN {X 0,Y 72.239,Z 834.42,A -85,B 0,C 180,E1 -28565.705,E2 -28565.705} C_VEL
LIN {X 0,Y 80.14,Z 835.472,A -85,B 0,C 180,E1 -28574.545,E2 -28574.545} C_VEL
LIN {X 0,Y 89.705,Z 835.241,A -85,B 0,C 180,E1 -28581.57,E2 -28581.57} C_VEL
LIN {X 0,Y 100.534,Z 833.737,A -85,B 0,C 180,E1 -28587.014,E2 -28587.014} C_VEL
LIN {X 0,Y 106.309,Z 832.495,A -85,B 0,C 180,E1 -28589.243,E2 -28589.243} C_VEL
LIN {X 0,Y 118.419,Z 828.929,A -85,B 0,C 180,E1 -28592.893,E2 -28592.893} C_VEL
LIN {X 0,Y 121.715,Z 827.766,A -85,B 0,C 180,E1 -28593.694,E2 -28593.694} C_VEL
LIN {X 0,Y 123.066,Z 827.168,A -85,B 0,C 180,E1 -28594.615,E2 -28594.615} C_VEL
LIN {X 0,Y 111.966,Z 830.232,A -85,B 0,C 180,E1 -28597.875,E2 -28597.875} C_VEL
LIN {X 0,Y 104.272,Z 831.621,A -85,B 0,C 180,E1 -28600.653,E2 -28600.653} C_VEL
LIN {X 0,Y 94.531,Z 832.546,A -85,B 0,C 180,E1 -28605.108,E2 -28605.108} C_VEL
LIN {X 0,Y 85.435,Z 832.376,A -85,B 0,C 180,E1 -28610.765,E2 -28610.765} C_VEL
LIN {X 0,Y 77.359,Z 831.071,A -85,B 0,C 180,E1 -28617.764,E2 -28617.764} C_VEL
LIN {X 0,Y 71.855,Z 829.109,A -85,B 0,C 180,E1 -28624.541,E2 -28624.541} C_VEL
LIN {X 0,Y 68.699,Z 827.736,A -85,B 0,C 180,E1 -28628.451,E2 -28628.451} C_VEL
LIN {X 0,Y 62.708,Z 824.725,A -85,B 0,C 180,E1 -28634.824,E2 -28634.824} C_VEL
LIN {X 0,Y 57.661,Z 820.972,A -85,B 0,C 180,E1 -28642.172,E2 -28642.172} C_VEL
LIN {X 0,Y 56.177,Z 818.37,A -85,B 0,C 180,E1 -28647.365,E2 -28647.365} C_VEL
LIN {X 0,Y 55.903,Z 812.168,A -85,B 0,C 180,E1 -28658.945,E2 -28658.945} C_VEL
LIN {X 0,Y 56.907,Z 806.27,A -85,B 0,C 180,E1 -28667.816,E2 -28667.816} C_VEL
LIN {X 0,Y 58.968,Z 798.928,A -85,B 0,C 180,E1 -28676.54,E2 -28676.54} C_VEL
LIN {X 0,Y 62.124,Z 789.788,A -85,B 0,C 180,E1 -28684.826,E2 -28684.826} C_VEL
LIN {X 0,Y 66.423,Z 778.577,A -85,B 0,C 180,E1 -28692.222,E2 -28692.222} C_VEL
LIN {X 0,Y 70.561,Z 766.931,A -85,B 0,C 180,E1 -28697.701,E2 -28697.701} C_VEL
LIN {X 0,Y 74.544,Z 754.425,A -85,B 0,C 180,E1 -28701.863,E2 -28701.863} C_VEL
LIN {X 0,Y 77.856,Z 741.68,A -85,B 0,C 180,E1 -28704.827,E2 -28704.827} C_VEL
LIN {X 0,Y 80.468,Z 727.681,A -85,B 0,C 180,E1 -28707.036,E2 -28707.036} C_VEL
LIN {X 0,Y 85.144,Z 690.441,A -85,B 0,C 180,E1 -28710.458,E2 -28710.458} C_VEL
LIN {X 0,Y 83.471,Z 684.867,A -85,B 0,C 180,E1 -28712.119,E2 -28712.119} C_VEL
LIN {X 0,Y 78.497,Z 671.493,A -85,B 0,C 180,E1 -28717.06,E2 -28717.06} C_VEL
LIN {X 0,Y 74.463,Z 662.26,A -85,B 0,C 180,E1 -28721.589,E2 -28721.589} C_VEL
LIN {X 0,Y 70.062,Z 655.065,A -85,B 0,C 180,E1 -28726.812,E2 -28726.812} C_VEL
LIN {X 0,Y 68.256,Z 652.408,A -85,B 0,C 180,E1 -28729.231,E2 -28729.231} C_VEL
LIN {X 0,Y 65.487,Z 648.456,A -85,B 0,C 180,E1 -28733.477,E2 -28733.477} C_VEL
LIN {X 0,Y 63.074,Z 645.611,A -85,B 0,C 180,E1 -28737.643,E2 -28737.643} C_VEL
LIN {X 0,Y 62.04,Z 643.646,A -85,B 0,C 180,E1 -28739.898,E2 -28739.898} C_VEL
LIN {X 0,Y 59.183,Z 641.315,A -85,B 0,C 180,E1 -28746.304,E2 -28746.304} C_VEL
LIN {X 0,Y 58.272,Z 639.128,A -85,B 0,C 180,E1 -28749.599,E2 -28749.599} C_VEL
LIN {X 0,Y 58.18,Z 638.229,A -85,B 0,C 180,E1 -28750.449,E2 -28750.449} C_VEL
LIN {X 0,Y 58.016,Z 638.231,A -85,B 0,C 180,E1 -28756.632,E2 -28756.632} C_VEL
LIN {X 0,Y 58.037,Z 638.191,A -85,B 0,C 180,E1 -28762.738,E2 -28762.738} C_VEL
LIN {X 0,Y 58.164,Z 638.206,A -85,B 0,C 180,E1 -28767.773,E2 -28767.773} C_VEL
LIN {X 0,Y 58.157,Z 638.236,A -85,B 0,C 180,E1 -28771.094,E2 -28771.094} C_VEL
LIN {X 0,Y 58.502,Z 638.136,A -85,B 0,C 180,E1 -28783.983,E2 -28783.983} C_VEL
LIN {X 0,Y 58.808,Z 638.158,A -85,B 0,C 180,E1 -28793.137,E2 -28793.137} C_VEL
LIN {X 0,Y 58.96,Z 638.205,A -85,B 0,C 180,E1 -28795.514,E2 -28795.514} C_VEL
LIN {X 0,Y 59.788,Z 640.237,A -85,B 0,C 180,E1 -28798.317,E2 -28798.317} C_VEL
LIN {X 0,Y 62.249,Z 643.248,A -85,B 0,C 180,E1 -28804.047,E2 -28804.047} C_VEL
LIN {X 0,Y 62.849,Z 643.875,A -85,B 0,C 180,E1 -28805.214,E2 -28805.214} C_VEL
LIN {X 0,Y 64.579,Z 647.086,A -85,B 0,C 180,E1 -28808.725,E2 -28808.725} C_VEL
LIN {X 0,Y 65.726,Z 648.533,A -85,B 0,C 180,E1 -28810.63,E2 -28810.63} C_VEL
LIN {X 0,Y 67.996,Z 652.319,A -85,B 0,C 180,E1 -28814.208,E2 -28814.208} C_VEL
LIN {X 0,Y 72.325,Z 659.672,A -85,B 0,C 180,E1 -28819.934,E2 -28819.934} C_VEL
LIN {X 0,Y 76.754,Z 668.762,A -85,B 0,C 180,E1 -28825.056,E2 -28825.056} C_VEL
LIN {X 0,Y 78.376,Z 672.826,A -85,B 0,C 180,E1 -28826.818,E2 -28826.818} C_VEL
LIN {X 0,Y 82.108,Z 686.084,A -85,B 0,C 180,E1 -28831.104,E2 -28831.104} C_VEL
LIN {X 0,Y 84.164,Z 694.962,A -85,B 0,C 180,E1 -28833.5,E2 -28833.5} C_VEL
LIN {X 0,Y 84.173,Z 704.481,A -85,B 0,C 180,E1 -28834.892,E2 -28834.892} C_VEL
LIN {X 0,Y 80.268,Z 736.48,A -85,B 0,C 180,E1 -28837.992,E2 -28837.992} C_VEL
LIN {X 0,Y 77.532,Z 750.589,A -85,B 0,C 180,E1 -28840.24,E2 -28840.24} C_VEL
LIN {X 0,Y 74.415,Z 762.147,A -85,B 0,C 180,E1 -28842.943,E2 -28842.943} C_VEL
LIN {X 0,Y 70.123,Z 775.369,A -85,B 0,C 180,E1 -28847.42,E2 -28847.42} C_VEL
LIN {X 0,Y 66.315,Z 785.78,A -85,B 0,C 180,E1 -28852.448,E2 -28852.448} C_VEL
LIN {X 0,Y 62.439,Z 796.313,A -85,B 0,C 180,E1 -28859.561,E2 -28859.561} C_VEL
LIN {X 0,Y 59.587,Z 804.925,A -85,B 0,C 180,E1 -28867.453,E2 -28867.453} C_VEL
LIN {X 0,Y 57.669,Z 812.936,A -85,B 0,C 180,E1 -28877.152,E2 -28877.152} C_VEL
LIN {X 0,Y 57.317,Z 818.965,A -85,B 0,C 180,E1 -28886.478,E2 -28886.478} C_VEL
LIN {X 0,Y 57.526,Z 822.639,A -85,B 0,C 180,E1 -28893.494,E2 -28893.494} C_VEL
LIN {X 0,Y 57.601,Z 826.781,A -85,B 0,C 180,E1 -28904.116,E2 -28904.116} C_VEL
LIN {X 0,Y 60.541,Z 830.804,A -85,B 0,C 180,E1 -28917.66,E2 -28917.66} C_VEL
LIN {X 0,Y 66.632,Z 833.454,A -85,B 0,C 180,E1 -28929.252,E2 -28929.252} C_VEL
LIN {X 0,Y 75.245,Z 834.82,A -85,B 0,C 180,E1 -28938.34,E2 -28938.34} C_VEL
LIN {X 0,Y 85.468,Z 834.895,A -85,B 0,C 180,E1 -28945.305,E2 -28945.305} C_VEL
LIN {X 0,Y 96.858,Z 833.7,A -85,B 0,C 180,E1 -28950.533,E2 -28950.533} C_VEL
LIN {X 0,Y 102.863,Z 832.622,A -85,B 0,C 180,E1 -28952.639,E2 -28952.639} C_VEL
LIN {X 0,Y 109.086,Z 831.203,A -85,B 0,C 180,E1 -28954.407,E2 -28954.407} C_VEL
LIN {X 0,Y 104.095,Z 832.032,A -85,B 0,C 180,E1 -28956.102,E2 -28956.102} C_VEL
LIN {X 0,Y 96.87,Z 832.849,A -85,B 0,C 180,E1 -28958.73,E2 -28958.73} C_VEL
LIN {X 0,Y 88.389,Z 833.128,A -85,B 0,C 180,E1 -28962.565,E2 -28962.565} C_VEL
LIN {X 0,Y 77.364,Z 832.248,A -85,B 0,C 180,E1 -28969.531,E2 -28969.531} C_VEL
LIN {X 0,Y 70.463,Z 830.648,A -85,B 0,C 180,E1 -28975.783,E2 -28975.783} C_VEL
LIN {X 0,Y 62.714,Z 827.19,A -85,B 0,C 180,E1 -28986.433,E2 -28986.433} C_VEL
LIN {X 0,Y 57.812,Z 822.364,A -85,B 0,C 180,E1 -28998.594,E2 -28998.594} C_VEL
LIN {X 0,Y 56.177,Z 818.37,A -85,B 0,C 180,E1 -29007.365,E2 -29007.365} C_VEL
LIN {X 0,Y 55.141,Z 815.623,A -85,B 0,C 180,E1 -29012.606,E2 -29012.606} C_VEL
LIN {X 0,Y 53.589,Z 812.547,A -85,B 0,C 180,E1 -29017.701,E2 -29017.701} C_VEL
LIN {X 0,Y 50.957,Z 805.624,A -85,B 0,C 180,E1 -29028.076,E2 -29028.076} C_VEL
LIN {X 0,Y 50.938,Z 801.821,A -85,B 0,C 180,E1 -29033.316,E2 -29033.316} C_VEL
LIN {X 0,Y 51.258,Z 800.507,A -85,B 0,C 180,E1 -29035.001,E2 -29035.001} C_VEL
LIN {X 0,Y 54.423,Z 791.598,A -85,B 0,C 180,E1 -29044.68,E2 -29044.68} C_VEL
LIN {X 0,Y 58.787,Z 780.711,A -85,B 0,C 180,E1 -29053.017,E2 -29053.017} C_VEL
LIN {X 0,Y 63.328,Z 768.942,A -85,B 0,C 180,E1 -29059.341,E2 -29059.341} C_VEL
LIN {X 0,Y 67.77,Z 756.043,A -85,B 0,C 180,E1 -29064.054,E2 -29064.054} C_VEL
LIN {X 0,Y 71.21,Z 743.834,A -85,B 0,C 180,E1 -29067.172,E2 -29067.172} C_VEL
LIN {X 0,Y 74.099,Z 730.131,A -85,B 0,C 180,E1 -29069.517,E2 -29069.517} C_VEL
LIN {X 0,Y 77.353,Z 706.191,A -85,B 0,C 180,E1 -29071.979,E2 -29071.979} C_VEL
LIN {X 0,Y 79.192,Z 691.423,A -85,B 0,C 180,E1 -29073.349,E2 -29073.349} C_VEL
LIN {X 0,Y 74.232,Z 676.755,A -85,B 0,C 180,E1 -29079.011,E2 -29079.011} C_VEL
LIN {X 0,Y 70.135,Z 666.811,A -85,B 0,C 180,E1 -29084.227,E2 -29084.227} C_VEL
LIN {X 0,Y 65.482,Z 658.74,A -85,B 0,C 180,E1 -29090.759,E2 -29090.759} C_VEL
LIN {X 0,Y 62.279,Z 654.209,A -85,B 0,C 180,E1 -29096.213,E2 -29096.213} C_VEL
LIN {X 0,Y 60.009,Z 651.025,A -85,B 0,C 180,E1 -29100.849,E2 -29100.849} C_VEL
LIN {X 0,Y 59.452,Z 649.999,A -85,B 0,C 180,E1 -29102.241,E2 -29102.241} C_VEL
LIN {X 0,Y 56.953,Z 647.501,A -85,B 0,C 180,E1 -29108.943,E2 -29108.943} C_VEL
LIN {X 0,Y 55.953,Z 645.023,A -85,B 0,C 180,E1 -29113.253,E2 -29113.253} C_VEL
LIN {X 0,Y 53.614,Z 643.664,A -85,B 0,C 180,E1 -29128.377,E2 -29128.377} C_VEL
LIN {X 0,Y 54.997,Z 644.221,A -85,B 0,C 180,E1 -29146.232,E2 -29146.232} C_VEL
LIN {X 0,Y 56.927,Z 645.153,A -85,B 0,C 180,E1 -29153.577,E2 -29153.577} C_VEL
LIN {X 0,Y 59.686,Z 649.439,A -85,B 0,C 180,E1 -29161.688,E2 -29161.688} C_VEL
LIN {X 0,Y 62.74,Z 654.638,A -85,B 0,C 180,E1 -29168.353,E2 -29168.353} C_VEL
LIN {X 0,Y 66.83,Z 661.788,A -85,B 0,C 180,E1 -29175.228,E2 -29175.228} C_VEL
LIN {X 0,Y 70.407,Z 668.977,A -85,B 0,C 180,E1 -29180.18,E2 -29180.18} C_VEL
LIN {X 0,Y 73.252,Z 675.83,A -85,B 0,C 180,E1 -29183.855,E2 -29183.855} C_VEL
LIN {X 0,Y 76.618,Z 688.595,A -85,B 0,C 180,E1 -29188.415,E2 -29188.415} C_VEL
LIN {X 0,Y 78.374,Z 696.081,A -85,B 0,C 180,E1 -29190.665,E2 -29190.665} C_VEL
LIN {X 0,Y 78.311,Z 705.164,A -85,B 0,C 180,E1 -29192.084,E2 -29192.084} C_VEL
LIN {X 0,Y 74.276,Z 736.052,A -85,B 0,C 180,E1 -29195.179,E2 -29195.179} C_VEL
LIN {X 0,Y 71.365,Z 750.211,A -85,B 0,C 180,E1 -29197.537,E2 -29197.537} C_VEL
LIN {X 0,Y 68.076,Z 761.794,A -85,B 0,C 180,E1 -29200.404,E2 -29200.404} C_VEL
LIN {X 0,Y 63.536,Z 774.9,A -85,B 0,C 180,E1 -29205.147,E2 -29205.147} C_VEL
LIN {X 0,Y 59.514,Z 785.306,A -85,B 0,C 180,E1 -29210.591,E2 -29210.591} C_VEL
LIN {X 0,Y 55.761,Z 794.879,A -85,B 0,C 180,E1 -29217.602,E2 -29217.602} C_VEL
LIN {X 0,Y 52.692,Z 803.653,A -85,B 0,C 180,E1 -29226.404,E2 -29226.404} C_VEL
LIN {X 0,Y 50.818,Z 810.977,A -85,B 0,C 180,E1 -29236.145,E2 -29236.145} C_VEL
LIN {X 0,Y 50.429,Z 817.911,A -85,B 0,C 180,E1 -29247.995,E2 -29247.995} C_VEL
LIN {X 0,Y 50.64,Z 820.754,A -85,B 0,C 180,E1 -29253.97,E2 -29253.97} C_VEL
LIN {X 0,Y 50.806,Z 824.611,A -85,B 0,C 180,E1 -29264.456,E2 -29264.456} C_VEL
LIN {X 0,Y 53.204,Z 828.52,A -85,B 0,C 180,E1 -29277.529,E2 -29277.529} C_VEL
LIN {X 0,Y 57.515,Z 831.11,A -85,B 0,C 180,E1 -29287.65,E2 -29287.65} C_VEL
LIN {X 0,Y 65.849,Z 833.39,A -85,B 0,C 180,E1 -29298.329,E2 -29298.329} C_VEL
LIN {X 0,Y 76.013,Z 834.391,A -85,B 0,C 180,E1 -29306.306,E2 -29306.306} C_VEL
LIN {X 0,Y 87.502,Z 834.172,A -85,B 0,C 180,E1 -29312.056,E2 -29312.056} C_VEL
LIN {X 0,Y 93.568,Z 833.595,A -85,B 0,C 180,E1 -29314.323,E2 -29314.323} C_VEL
LIN {X 0,Y 92.886,Z 833.554,A -85,B 0,C 180,E1 -29315.211,E2 -29315.211} C_VEL
LIN {X 0,Y 81.899,Z 833.448,A -85,B 0,C 180,E1 -29319.924,E2 -29319.924} C_VEL
LIN {X 0,Y 72.569,Z 832.318,A -85,B 0,C 180,E1 -29325.547,E2 -29325.547} C_VEL
LIN {X 0,Y 63.408,Z 829.914,A -85,B 0,C 180,E1 -29333.635,E2 -29333.635} C_VEL
LIN {X 0,Y 56.321,Z 826.483,A -85,B 0,C 180,E1 -29343.492,E2 -29343.492} C_VEL
LIN {X 0,Y 51.181,Z 821.701,A -85,B 0,C 180,E1 -29356.042,E2 -29356.042} C_VEL
LIN {X 0,Y 48.897,Z 815.404,A -85,B 0,C 180,E1 -29370.433,E2 -29370.433} C_VEL
LIN {X 0,Y 49.169,Z 809.183,A -85,B 0,C 180,E1 -29382.251,E2 -29382.251} C_VEL
LIN {X 0,Y 51.258,Z 800.507,A -85,B 0,C 180,E1 -29395.001,E2 -29395.001} C_VEL
LIN {X 0,Y 51.939,Z 796.525,A -85,B 0,C 180,E1 -29399.783,E2 -29399.783} C_VEL
LIN {X 0,Y 51.803,Z 789.404,A -85,B 0,C 180,E1 -29407.418,E2 -29407.418} C_VEL
LIN {X 0,Y 52.203,Z 781.764,A -85,B 0,C 180,E1 -29414.478,E2 -29414.478} C_VEL
LIN {X 0,Y 53.638,Z 776.94,A -85,B 0,C 180,E1 -29417.924,E2 -29417.924} C_VEL
LIN {X 0,Y 58.38,Z 765.147,A -85,B 0,C 180,E1 -29423.965,E2 -29423.965} C_VEL
LIN {X 0,Y 62.449,Z 753.502,A -85,B 0,C 180,E1 -29428.041,E2 -29428.041} C_VEL
LIN {X 0,Y 66.174,Z 740.294,A -85,B 0,C 180,E1 -29431.141,E2 -29431.141} C_VEL
LIN {X 0,Y 68.881,Z 726.669,A -85,B 0,C 180,E1 -29433.289,E2 -29433.289} C_VEL
LIN {X 0,Y 73.442,Z 692.97,A -85,B 0,C 180,E1 -29436.576,E2 -29436.576} C_VEL
LIN {X 0,Y 68.874,Z 678.991,A -85,B 0,C 180,E1 -29442.738,E2 -29442.738} C_VEL
LIN {X 0,Y 65.879,Z 671.314,A -85,B 0,C 180,E1 -29447.22,E2 -29447.22} C_VEL
LIN {X 0,Y 62.147,Z 664.324,A -85,B 0,C 180,E1 -29453.445,E2 -29453.445} C_VEL
LIN {X 0,Y 59.309,Z 660.059,A -85,B 0,C 180,E1 -29458.925,E2 -29458.925} C_VEL
LIN {X 0,Y 56.896,Z 656.264,A -85,B 0,C 180,E1 -29464.979,E2 -29464.979} C_VEL
LIN {X 0,Y 54.685,Z 653.402,A -85,B 0,C 180,E1 -29472.375,E2 -29472.375} C_VEL
LIN {X 0,Y 54.092,Z 651.817,A -85,B 0,C 180,E1 -29475.487,E2 -29475.487} C_VEL
LIN {X 0,Y 52.423,Z 650.708,A -85,B 0,C 180,E1 -29487.572,E2 -29487.572} C_VEL
LIN {X 0,Y 53.432,Z 651.101,A -85,B 0,C 180,E1 -29504.749,E2 -29504.749} C_VEL
LIN {X 0,Y 55.114,Z 652.072,A -85,B 0,C 180,E1 -29511.991,E2 -29511.991} C_VEL
LIN {X 0,Y 57.603,Z 656.425,A -85,B 0,C 180,E1 -29520.329,E2 -29520.329} C_VEL
LIN {X 0,Y 59.914,Z 660.822,A -85,B 0,C 180,E1 -29525.998,E2 -29525.998} C_VEL
LIN {X 0,Y 63.277,Z 667.254,A -85,B 0,C 180,E1 -29532.604,E2 -29532.604} C_VEL
LIN {X 0,Y 66.181,Z 673.58,A -85,B 0,C 180,E1 -29537.327,E2 -29537.327} C_VEL
LIN {X 0,Y 68.6,Z 679.82,A -85,B 0,C 180,E1 -29540.897,E2 -29540.897} C_VEL
LIN {X 0,Y 71.589,Z 692.379,A -85,B 0,C 180,E1 -29545.786,E2 -29545.786} C_VEL
LIN {X 0,Y 72.796,Z 698.341,A -85,B 0,C 180,E1 -29547.714,E2 -29547.714} C_VEL
LIN {X 0,Y 72.576,Z 705.702,A -85,B 0,C 180,E1 -29548.896,E2 -29548.896} C_VEL
LIN {X 0,Y 68.401,Z 735.759,A -85,B 0,C 180,E1 -29551.984,E2 -29551.984} C_VEL
LIN {X 0,Y 65.442,Z 749.488,A -85,B 0,C 180,E1 -29554.342,E2 -29554.342} C_VEL
LIN {X 0,Y 61.898,Z 761.314,A -85,B 0,C 180,E1 -29557.354,E2 -29557.354} C_VEL
LIN {X 0,Y 57.09,Z 774.431,A -85,B 0,C 180,E1 -29562.375,E2 -29562.375} C_VEL
LIN {X 0,Y 52.325,Z 785.981,A -85,B 0,C 180,E1 -29569.086,E2 -29569.086} C_VEL
LIN {X 0,Y 48.426,Z 795.354,A -85,B 0,C 180,E1 -29577.018,E2 -29577.018} C_VEL
LIN {X 0,Y 45.337,Z 803.904,A -85,B 0,C 180,E1 -29587.188,E2 -29587.188} C_VEL
LIN {X 0,Y 43.494,Z 812.204,A -85,B 0,C 180,E1 -29600.691,E2 -29600.691} C_VEL
LIN {X 0,Y 43.585,Z 816.75,A -85,B 0,C 180,E1 -29609.99,E2 -29609.99} C_VEL
LIN {X 0,Y 43.794,Z 818.735,A -85,B 0,C 180,E1 -29614.592,E2 -29614.592} C_VEL
LIN {X 0,Y 43.98,Z 821.882,A -85,B 0,C 180,E1 -29623.58,E2 -29623.58} C_VEL
LIN {X 0,Y 45.933,Z 825.885,A -85,B 0,C 180,E1 -29637.313,E2 -29637.313} C_VEL
LIN {X 0,Y 52.142,Z 829.781,A -85,B 0,C 180,E1 -29652.359,E2 -29652.359} C_VEL
LIN {X 0,Y 61.385,Z 832.39,A -85,B 0,C 180,E1 -29663.255,E2 -29663.255} C_VEL
LIN {X 0,Y 72.332,Z 833.717,A -85,B 0,C 180,E1 -29670.97,E2 -29670.97} C_VEL
LIN {X 0,Y 78.273,Z 833.934,A -85,B 0,C 180,E1 -29673.868,E2 -29673.868} C_VEL
LIN {X 0,Y 78.594,Z 833.809,A -85,B 0,C 180,E1 -29675.415,E2 -29675.415} C_VEL
LIN {X 0,Y 66.438,Z 831.945,A -85,B 0,C 180,E1 -29682.162,E2 -29682.162} C_VEL
LIN {X 0,Y 57.016,Z 829.114,A -85,B 0,C 180,E1 -29690.393,E2 -29690.393} C_VEL
LIN {X 0,Y 49.205,Z 825.045,A -85,B 0,C 180,E1 -29701.523,E2 -29701.523} C_VEL
LIN {X 0,Y 43.853,Z 819.641,A -85,B 0,C 180,E1 -29715.972,E2 -29715.972} C_VEL
LIN {X 0,Y 41.811,Z 812.737,A -85,B 0,C 180,E1 -29732.831,E2 -29732.831} C_VEL
LIN {X 0,Y 42.438,Z 806.473,A -85,B 0,C 180,E1 -29745.462,E2 -29745.462} C_VEL
LIN {X 0,Y 44.785,Z 798.261,A -85,B 0,C 180,E1 -29758.224,E2 -29758.224} C_VEL
LIN {X 0,Y 48.769,Z 788.15,A -85,B 0,C 180,E1 -29769.501,E2 -29769.501} C_VEL
LIN {X 0,Y 53.638,Z 776.94,A -85,B 0,C 180,E1 -29777.924,E2 -29777.924} C_VEL
LIN {X 0,Y 55.079,Z 772.086,A -85,B 0,C 180,E1 -29780.98,E2 -29780.98} C_VEL
LIN {X 0,Y 55.867,Z 763.651,A -85,B 0,C 180,E1 -29786.276,E2 -29786.276} C_VEL
LIN {X 0,Y 56.61,Z 754.822,A -85,B 0,C 180,E1 -29791.016,E2 -29791.016} C_VEL
LIN {X 0,Y 57.877,Z 749.267,A -85,B 0,C 180,E1 -29792.969,E2 -29792.969} C_VEL
LIN {X 0,Y 61.507,Z 735.9,A -85,B 0,C 180,E1 -29795.752,E2 -29795.752} C_VEL
LIN {X 0,Y 63.987,Z 722.608,A -85,B 0,C 180,E1 -29797.553,E2 -29797.553} C_VEL
LIN {X 0,Y 67.908,Z 694.725,A -85,B 0,C 180,E1 -29800.278,E2 -29800.278} C_VEL
LIN {X 0,Y 64.292,Z 682.76,A -85,B 0,C 180,E1 -29806.1,E2 -29806.1} C_VEL
LIN {X 0,Y 61.849,Z 675.784,A -85,B 0,C 180,E1 -29810.601,E2 -29810.601} C_VEL
LIN {X 0,Y 58.793,Z 669.734,A -85,B 0,C 180,E1 -29816.564,E2 -29816.564} C_VEL
LIN {X 0,Y 56.462,Z 665.892,A -85,B 0,C 180,E1 -29821.944,E2 -29821.944} C_VEL
LIN {X 0,Y 54.631,Z 662.628,A -85,B 0,C 180,E1 -29827.521,E2 -29827.521} C_VEL
LIN {X 0,Y 52.66,Z 659.513,A -85,B 0,C 180,E1 -29835.575,E2 -29835.575} C_VEL
LIN {X 0,Y 52.314,Z 658.587,A -85,B 0,C 180,E1 -29837.802,E2 -29837.802} C_VEL
LIN {X 0,Y 51.236,Z 657.778,A -85,B 0,C 180,E1 -29846.725,E2 -29846.725} C_VEL
LIN {X 0,Y 51.727,Z 657.946,A -85,B 0,C 180,E1 -29862.028,E2 -29862.028} C_VEL
LIN {X 0,Y 53.29,Z 658.752,A -85,B 0,C 180,E1 -29869.939,E2 -29869.939} C_VEL
LIN {X 0,Y 55.18,Z 662.668,A -85,B 0,C 180,E1 -29877.666,E2 -29877.666} C_VEL
LIN {X 0,Y 57.095,Z 666.826,A -85,B 0,C 180,E1 -29883.309,E2 -29883.309} C_VEL
LIN {X 0,Y 59.882,Z 672.659,A -85,B 0,C 180,E1 -29889.674,E2 -29889.674} C_VEL
LIN {X 0,Y 62.39,Z 678.944,A -85,B 0,C 180,E1 -29894.638,E2 -29894.638} C_VEL
LIN {X 0,Y 63.992,Z 683.569,A -85,B 0,C 180,E1 -29897.508,E2 -29897.508} C_VEL
LIN {X 0,Y 66.545,Z 695.373,A -85,B 0,C 180,E1 -29902.462,E2 -29902.462} C_VEL
LIN {X 0,Y 67.415,Z 699.871,A -85,B 0,C 180,E1 -29904.128,E2 -29904.128} C_VEL
LIN {X 0,Y 67.145,Z 705.947,A -85,B 0,C 180,E1 -29905.164,E2 -29905.164} C_VEL
LIN {X 0,Y 62.8,Z 735.35,A -85,B 0,C 180,E1 -29908.187,E2 -29908.187} C_VEL
LIN {X 0,Y 59.689,Z 748.979,A -85,B 0,C 180,E1 -29910.558,E2 -29910.558} C_VEL
LIN {X 0,Y 55.942,Z 760.773,A -85,B 0,C 180,E1 -29913.651,E2 -29913.651} C_VEL
LIN {X 0,Y 50.809,Z 773.807,A -85,B 0,C 180,E1 -29918.904,E2 -29918.904} C_VEL
LIN {X 0,Y 46.215,Z 784.188,A -85,B 0,C 180,E1 -29925.292,E2 -29925.292} C_VEL
LIN {X 0,Y 41.896,Z 793.727,A -85,B 0,C 180,E1 -29934.034,E2 -29934.034} C_VEL
LIN {X 0,Y 37.992,Z 804.033,A -85,B 0,C 180,E1 -29948.274,E2 -29948.274} C_VEL
LIN {X 0,Y 36.524,Z 812.174,A -85,B 0,C 180,E1 -29964.467,E2 -29964.467} C_VEL
LIN {X 0,Y 36.949,Z 816.601,A -85,B 0,C 180,E1 -29975.445,E2 -29975.445} C_VEL
LIN {X 0,Y 37.175,Z 818.442,A -85,B 0,C 180,E1 -29980.885,E2 -29980.885} C_VEL
LIN {X 0,Y 39.938,Z 824.156,A -85,B 0,C 180,E1 -30001.852,E2 -30001.852} C_VEL
LIN {X 0,Y 47.214,Z 828.409,A -85,B 0,C 180,E1 -30018.082,E2 -30018.082} C_VEL
LIN {X 0,Y 57.444,Z 831.296,A -85,B 0,C 180,E1 -30028.902,E2 -30028.902} C_VEL
LIN {X 0,Y 66.169,Z 832.612,A -85,B 0,C 180,E1 -30034.858,E2 -30034.858} C_VEL
LIN {X 0,Y 55.81,Z 829.931,A -85,B 0,C 180,E1 -30041.649,E2 -30041.649} C_VEL
LIN {X 0,Y 46.713,Z 826.136,A -85,B 0,C 180,E1 -30051.346,E2 -30051.346} C_VEL
LIN {X 0,Y 39.519,Z 821.093,A -85,B 0,C 180,E1 -30065.1,E2 -30065.1} C_VEL
LIN {X 0,Y 35.411,Z 814.593,A -85,B 0,C 180,E1 -30083.385,E2 -30083.385} C_VEL
LIN {X 0,Y 35.026,Z 807.776,A -85,B 0,C 180,E1 -30100.699,E2 -30100.699} C_VEL
LIN {X 0,Y 37.052,Z 799.735,A -85,B 0,C 180,E1 -30116.556,E2 -30116.556} C_VEL
LIN {X 0,Y 41.031,Z 789.926,A -85,B 0,C 180,E1 -30129.978,E2 -30129.978} C_VEL
LIN {X 0,Y 46.132,Z 779.042,A -85,B 0,C 180,E1 -30139.763,E2 -30139.763} C_VEL
LIN {X 0,Y 51.467,Z 766.729,A -85,B 0,C 180,E1 -30146.896,E2 -30146.896} C_VEL
LIN {X 0,Y 56.244,Z 754.262,A -85,B 0,C 180,E1 -30151.578,E2 -30151.578} C_VEL
LIN {X 0,Y 57.877,Z 749.267,A -85,B 0,C 180,E1 -30152.969,E2 -30152.969} C_VEL
LIN {X 0,Y 59.005,Z 743.726,A -85,B 0,C 180,E1 -30154.667,E2 -30154.667} C_VEL
LIN {X 0,Y 59.116,Z 734.466,A -85,B 0,C 180,E1 -30158.136,E2 -30158.136} C_VEL
LIN {X 0,Y 58.797,Z 725.032,A -85,B 0,C 180,E1 -30161.3,E2 -30161.3} C_VEL
LIN {X 0,Y 59.212,Z 719.204,A -85,B 0,C 180,E1 -30162.353,E2 -30162.353} C_VEL
LIN {X 0,Y 62.611,Z 696.461,A -85,B 0,C 180,E1 -30164.502,E2 -30164.502} C_VEL
LIN {X 0,Y 59.976,Z 686.623,A -85,B 0,C 180,E1 -30169.924,E2 -30169.924} C_VEL
LIN {X 0,Y 58.034,Z 680.32,A -85,B 0,C 180,E1 -30174.351,E2 -30174.351} C_VEL
LIN {X 0,Y 55.662,Z 675.21,A -85,B 0,C 180,E1 -30179.886,E2 -30179.886} C_VEL
LIN {X 0,Y 53.802,Z 671.691,A -85,B 0,C 180,E1 -30185.231,E2 -30185.231} C_VEL
LIN {X 0,Y 52.387,Z 668.82,A -85,B 0,C 180,E1 -30190.622,E2 -30190.622} C_VEL
LIN {X 0,Y 50.666,Z 665.394,A -85,B 0,C 180,E1 -30200.004,E2 -30200.004} C_VEL
LIN {X 0,Y 49.954,Z 664.743,A -85,B 0,C 180,E1 -30207.595,E2 -30207.595} C_VEL
LIN {X 0,Y 50.951,Z 665.1,A -85,B 0,C 180,E1 -30224.949,E2 -30224.949} C_VEL
LIN {X 0,Y 51.598,Z 665.619,A -85,B 0,C 180,E1 -30228.252,E2 -30228.252} C_VEL
LIN {X 0,Y 52.924,Z 668.933,A -85,B 0,C 180,E1 -30234.887,E2 -30234.887} C_VEL
LIN {X 0,Y 55.202,Z 674.581,A -85,B 0,C 180,E1 -30242.71,E2 -30242.71} C_VEL
LIN {X 0,Y 57.894,Z 681.488,A -85,B 0,C 180,E1 -30249.531,E2 -30249.531} C_VEL
LIN {X 0,Y 59.648,Z 687.323,A -85,B 0,C 180,E1 -30253.631,E2 -30253.631} C_VEL
LIN {X 0,Y 61.951,Z 700.154,A -85,B 0,C 180,E1 -30259.448,E2 -30259.448} C_VEL
LIN {X 0,Y 62.216,Z 702.295,A -85,B 0,C 180,E1 -30260.207,E2 -30260.207} C_VEL
LIN {X 0,Y 61.758,Z 707.52,A -85,B 0,C 180,E1 -30260.998,E2 -30260.998} C_VEL
LIN {X 0,Y 57.384,Z 735.096,A -85,B 0,C 180,E1 -30263.816,E2 -30263.816} C_VEL
LIN {X 0,Y 53.906,Z 749.24,A -85,B 0,C 180,E1 -30266.304,E2 -30266.304} C_VEL
LIN {X 0,Y 49.561,Z 761.68,A -85,B 0,C 180,E1 -30269.692,E2 -30269.692} C_VEL
LIN {X 0,Y 44.124,Z 774.473,A -85,B 0,C 180,E1 -30275.268,E2 -30275.268} C_VEL
LIN {X 0,Y 38.662,Z 785.729,A -85,B 0,C 180,E1 -30283.338,E2 -30283.338} C_VEL
LIN {X 0,Y 33.672,Z 796.04,A -85,B 0,C 180,E1 -30295.321,E2 -30295.321} C_VEL
LIN {X 0,Y 30.761,Z 803.632,A -85,B 0,C 180,E1 -30308.82,E2 -30308.82} C_VEL
LIN {X 0,Y 29.814,Z 812.072,A -85,B 0,C 180,E1 -30329.985,E2 -30329.985} C_VEL
LIN {X 0,Y 30.166,Z 814.321,A -85,B 0,C 180,E1 -30336.675,E2 -30336.675} C_VEL
LIN {X 0,Y 30.794,Z 817.508,A -85,B 0,C 180,E1 -30348.111,E2 -30348.111} C_VEL
LIN {X 0,Y 34.293,Z 822.368,A -85,B 0,C 180,E1 -30367.923,E2 -30367.923} C_VEL
LIN {X 0,Y 42.88,Z 826.857,A -85,B 0,C 180,E1 -30385.016,E2 -30385.016} C_VEL
LIN {X 0,Y 51.158,Z 829.411,A -85,B 0,C 180,E1 -30393.169,E2 -30393.169} C_VEL
LIN {X 0,Y 52.364,Z 829.628,A -85,B 0,C 180,E1 -30395.051,E2 -30395.051} C_VEL
LIN {X 0,Y 41.435,Z 825.123,A -85,B 0,C 180,E1 -30405.254,E2 -30405.254} C_VEL
LIN {X 0,Y 33.306,Z 819.664,A -85,B 0,C 180,E1 -30419.998,E2 -30419.998} C_VEL
LIN {X 0,Y 28.46,Z 812.599,A -85,B 0,C 180,E1 -30442.159,E2 -30442.159} C_VEL
LIN {X 0,Y 28.243,Z 805.295,A -85,B 0,C 180,E1 -30463.646,E2 -30463.646} C_VEL
LIN {X 0,Y 30.787,Z 797.091,A -85,B 0,C 180,E1 -30481.837,E2 -30481.837} C_VEL
LIN {X 0,Y 35.316,Z 787.43,A -85,B 0,C 180,E1 -30495.956,E2 -30495.956} C_VEL
LIN {X 0,Y 40.626,Z 777.1,A -85,B 0,C 180,E1 -30505.368,E2 -30505.368} C_VEL
LIN {X 0,Y 45.645,Z 766.35,A -85,B 0,C 180,E1 -30511.647,E2 -30511.647} C_VEL
LIN {X 0,Y 50.537,Z 754.368,A -85,B 0,C 180,E1 -30516.13,E2 -30516.13} C_VEL
LIN {X 0,Y 54.894,Z 740.604,A -85,B 0,C 180,E1 -30519.464,E2 -30519.464} C_VEL
LIN {X 0,Y 57.813,Z 728,A -85,B 0,C 180,E1 -30521.404,E2 -30521.404} C_VEL
LIN {X 0,Y 59.212,Z 719.204,A -85,B 0,C 180,E1 -30522.353,E2 -30522.353} C_VEL
LIN {X 0,Y 59.345,Z 715.314,A -85,B 0,C 180,E1 -30523.168,E2 -30523.168} C_VEL
LIN {X 0,Y 57.461,Z 703.059,A -85,B 0,C 180,E1 -30528.434,E2 -30528.434} C_VEL
LIN {X 0,Y 57.666,Z 699.168,A -85,B 0,C 180,E1 -30529.28,E2 -30529.28} C_VEL
LIN {X 0,Y 57.544,Z 697.492,A -85,B 0,C 180,E1 -30529.916,E2 -30529.916} C_VEL
LIN {X 0,Y 55.712,Z 689.68,A -85,B 0,C 180,E1 -30534.78,E2 -30534.78} C_VEL
LIN {X 0,Y 54.454,Z 685.04,A -85,B 0,C 180,E1 -30538.415,E2 -30538.415} C_VEL
LIN {X 0,Y 52.684,Z 680.58,A -85,B 0,C 180,E1 -30543.764,E2 -30543.764} C_VEL
LIN {X 0,Y 51.069,Z 676.938,A -85,B 0,C 180,E1 -30549.941,E2 -30549.941} C_VEL
LIN {X 0,Y 50.29,Z 675.121,A -85,B 0,C 180,E1 -30553.605,E2 -30553.605} C_VEL
LIN {X 0,Y 49.114,Z 672.189,A -85,B 0,C 180,E1 -30562.172,E2 -30562.172} C_VEL
LIN {X 0,Y 48.617,Z 671.683,A -85,B 0,C 180,E1 -30574.3,E2 -30574.3} C_VEL
LIN {X 0,Y 49.829,Z 672.191,A -85,B 0,C 180,E1 -30585.775,E2 -30585.775} C_VEL
LIN {X 0,Y 50.751,Z 675.116,A -85,B 0,C 180,E1 -30591.669,E2 -30591.669} C_VEL
LIN {X 0,Y 52.191,Z 679.66,A -85,B 0,C 180,E1 -30598.406,E2 -30598.406} C_VEL
LIN {X 0,Y 54.199,Z 685.692,A -85,B 0,C 180,E1 -30605.056,E2 -30605.056} C_VEL
LIN {X 0,Y 55.552,Z 690.941,A -85,B 0,C 180,E1 -30609.047,E2 -30609.047} C_VEL
LIN {X 0,Y 57.163,Z 702.119,A -85,B 0,C 180,E1 -30614.716,E2 -30614.716} C_VEL
LIN {X 0,Y 57.315,Z 704.431,A -85,B 0,C 180,E1 -30615.55,E2 -30615.55} C_VEL
LIN {X 0,Y 52.813,Z 732.85,A -85,B 0,C 180,E1 -30618.379,E2 -30618.379} C_VEL
LIN {X 0,Y 49.271,Z 746.926,A -85,B 0,C 180,E1 -30620.573,E2 -30620.573} C_VEL
LIN {X 0,Y 45.03,Z 759.025,A -85,B 0,C 180,E1 -30623.495,E2 -30623.495} C_VEL
LIN {X 0,Y 39.825,Z 770.764,A -85,B 0,C 180,E1 -30628.048,E2 -30628.048} C_VEL
LIN {X 0,Y 33.642,Z 782.648,A -85,B 0,C 180,E1 -30635.93,E2 -30635.93} C_VEL
LIN {X 0,Y 28.196,Z 792.639,A -85,B 0,C 180,E1 -30647.687,E2 -30647.687} C_VEL
LIN {X 0,Y 23.975,Z 801.851,A -85,B 0,C 180,E1 -30666.492,E2 -30666.492} C_VEL
LIN {X 0,Y 23.145,Z 810.714,A -85,B 0,C 180,E1 -30694.335,E2 -30694.335} C_VEL
LIN {X 0,Y 24.025,Z 813.976,A -85,B 0,C 180,E1 -30706.99,E2 -30706.99} C_VEL
LIN {X 0,Y 26.94,Z 818.612,A -85,B 0,C 180,E1 -30728.494,E2 -30728.494} C_VEL
LIN {X 0,Y 33.882,Z 822.978,A -85,B 0,C 180,E1 -30746.044,E2 -30746.044} C_VEL
LIN {X 0,Y 39.324,Z 825.232,A -85,B 0,C 180,E1 -30753.303,E2 -30753.303} C_VEL
LIN {X 0,Y 38.544,Z 824.785,A -85,B 0,C 180,E1 -30755.711,E2 -30755.711} C_VEL
LIN {X 0,Y 28.518,Z 818.873,A -85,B 0,C 180,E1 -30770.23,E2 -30770.23} C_VEL
LIN {X 0,Y 21.962,Z 811.36,A -85,B 0,C 180,E1 -30796.332,E2 -30796.332} C_VEL
LIN {X 0,Y 21.173,Z 804.7,A -85,B 0,C 180,E1 -30821.592,E2 -30821.592} C_VEL
LIN {X 0,Y 24.169,Z 795.759,A -85,B 0,C 180,E1 -30846.45,E2 -30846.45} C_VEL
LIN {X 0,Y 29.262,Z 786.228,A -85,B 0,C 180,E1 -30862.174,E2 -30862.174} C_VEL
LIN {X 0,Y 35.159,Z 775.788,A -85,B 0,C 180,E1 -30871.946,E2 -30871.946} C_VEL
LIN {X 0,Y 41.054,Z 763.943,A -85,B 0,C 180,E1 -30878.47,E2 -30878.47} C_VEL
LIN {X 0,Y 45.857,Z 752.532,A -85,B 0,C 180,E1 -30882.312,E2 -30882.312} C_VEL
LIN {X 0,Y 50.035,Z 739.958,A -85,B 0,C 180,E1 -30885.061,E2 -30885.061} C_VEL
LIN {X 0,Y 53.135,Z 726.813,A -85,B 0,C 180,E1 -30886.855,E2 -30886.855} C_VEL
LIN {X 0,Y 57.666,Z 699.168,A -85,B 0,C 180,E1 -30889.28,E2 -30889.28} C_VEL
LIN {X 0,Y 57.537,Z 696.638,A -85,B 0,C 180,E1 -30890.176,E2 -30890.176} C_VEL
LIN {X 0,Y 56.408,Z 694.206,A -85,B 0,C 180,E1 -30892.384,E2 -30892.384} C_VEL
LIN {X 0,Y 54.666,Z 692.33,A -85,B 0,C 180,E1 -30895.509,E2 -30895.509} C_VEL
LIN {X 0,Y 51.083,Z 688.827,A -85,B 0,C 180,E1 -30903.702,E2 -30903.702} C_VEL
LIN {X 0,Y 50.402,Z 687.047,A -85,B 0,C 180,E1 -30906.281,E2 -30906.281} C_VEL
LIN {X 0,Y 48.921,Z 683.092,A -85,B 0,C 180,E1 -30913.151,E2 -30913.151} C_VEL
LIN {X 0,Y 48.32,Z 681.412,A -85,B 0,C 180,E1 -30916.947,E2 -30916.947} C_VEL
LIN {X 0,Y 47.683,Z 679.029,A -85,B 0,C 180,E1 -30923.875,E2 -30923.875} C_VEL
LIN {X 0,Y 47.355,Z 678.656,A -85,B 0,C 180,E1 -30933.563,E2 -30933.563} C_VEL
LIN {X 0,Y 48.18,Z 678.976,A -85,B 0,C 180,E1 -30943.551,E2 -30943.551} C_VEL
LIN {X 0,Y 48.773,Z 681.491,A -85,B 0,C 180,E1 -30948.707,E2 -30948.707} C_VEL
LIN {X 0,Y 50.388,Z 688.147,A -85,B 0,C 180,E1 -30958.041,E2 -30958.041} C_VEL
LIN {X 0,Y 51.691,Z 693.974,A -85,B 0,C 180,E1 -30963.563,E2 -30963.563} C_VEL
LIN {X 0,Y 52.919,Z 705.277,A -85,B 0,C 180,E1 -30969.787,E2 -30969.787} C_VEL
LIN {X 0,Y 47.888,Z 734.208,A -85,B 0,C 180,E1 -30972.357,E2 -30972.357} C_VEL
LIN {X 0,Y 43.999,Z 748.223,A -85,B 0,C 180,E1 -30974.411,E2 -30974.411} C_VEL
LIN {X 0,Y 39.511,Z 759.73,A -85,B 0,C 180,E1 -30977.01,E2 -30977.01} C_VEL
LIN {X 0,Y 33.183,Z 772.607,A -85,B 0,C 180,E1 -30982.056,E2 -30982.056} C_VEL
LIN {X 0,Y 26.51,Z 783.968,A -85,B 0,C 180,E1 -30990.473,E2 -30990.473} C_VEL
LIN {X 0,Y 20.243,Z 794.142,A -85,B 0,C 180,E1 -31005.995,E2 -31005.995} C_VEL
LIN {X 0,Y 16.416,Z 802.446,A -85,B 0,C 180,E1 -31031.244,E2 -31031.244} C_VEL
LIN {X 0,Y 16.729,Z 809.275,A -85,B 0,C 180,E1 -31062.099,E2 -31062.099} C_VEL
LIN {X 0,Y 17.74,Z 811.514,A -85,B 0,C 180,E1 -31073.312,E2 -31073.312} C_VEL
LIN {X 0,Y 22.974,Z 817.04,A -85,B 0,C 180,E1 -31102.276,E2 -31102.276} C_VEL
LIN {X 0,Y 25.005,Z 818.302,A -85,B 0,C 180,E1 -31107.444,E2 -31107.444} C_VEL
LIN {X 0,Y 27.019,Z 819.322,A -85,B 0,C 180,E1 -31113.989,E2 -31113.989} C_VEL
LIN {X 0,Y 18.058,Z 812.63,A -85,B 0,C 180,E1 -31134.408,E2 -31134.408} C_VEL
LIN {X 0,Y 14.168,Z 805.392,A -85,B 0,C 180,E1 -31169.734,E2 -31169.734} C_VEL
LIN {X 0,Y 16.021,Z 797.774,A -85,B 0,C 180,E1 -31204.01,E2 -31204.01} C_VEL
LIN {X 0,Y 21.144,Z 789.013,A -85,B 0,C 180,E1 -31225.656,E2 -31225.656} C_VEL
LIN {X 0,Y 27.635,Z 778.823,A -85,B 0,C 180,E1 -31237.596,E2 -31237.596} C_VEL
LIN {X 0,Y 34.614,Z 766.555,A -85,B 0,C 180,E1 -31244.827,E2 -31244.827} C_VEL
LIN {X 0,Y 40.198,Z 754.642,A -85,B 0,C 180,E1 -31248.662,E2 -31248.662} C_VEL
LIN {X 0,Y 44.713,Z 742.185,A -85,B 0,C 180,E1 -31251.197,E2 -31251.197} C_VEL
LIN {X 0,Y 48.329,Z 728.446,A -85,B 0,C 180,E1 -31252.903,E2 -31252.903} C_VEL
LIN {X 0,Y 53.195,Z 700.065,A -85,B 0,C 180,E1 -31255.212,E2 -31255.212} C_VEL
LIN {X 0,Y 51.904,Z 693.133,A -85,B 0,C 180,E1 -31260.067,E2 -31260.067} C_VEL
LIN {X 0,Y 51.132,Z 689.531,A -85,B 0,C 180,E1 -31263.259,E2 -31263.259} C_VEL
LIN {X 0,Y 50.402,Z 687.047,A -85,B 0,C 180,E1 -31266.281,E2 -31266.281} C_VEL
LIN {X 0,Y 49.68,Z 685.382,A -85,B 0,C 180,E1 -31269.287,E2 -31269.287} C_VEL
LIN {X 0,Y 48.389,Z 684.543,A -85,B 0,C 180,E1 -31274.324,E2 -31274.324} C_VEL
LIN {X 0,Y 46.088,Z 685.706,A -85,B 0,C 180,E1 -31291.222,E2 -31291.222} C_VEL
LIN {X 0,Y 46.681,Z 686.035,A -85,B 0,C 180,E1 -31302.111,E2 -31302.111} C_VEL
LIN {X 0,Y 47.48,Z 691.702,A -85,B 0,C 180,E1 -31311.062,E2 -31311.062} C_VEL
LIN {X 0,Y 48.157,Z 695.976,A -85,B 0,C 180,E1 -31316.081,E2 -31316.081} C_VEL
LIN {X 0,Y 48.446,Z 698.57,A -85,B 0,C 180,E1 -31318.289,E2 -31318.289} C_VEL
LIN {X 0,Y 48.886,Z 706.76,A -85,B 0,C 180,E1 -31323.172,E2 -31323.172} C_VEL
LIN {X 0,Y 43.902,Z 733.896,A -85,B 0,C 180,E1 -31325.038,E2 -31325.038} C_VEL
LIN {X 0,Y 39.8,Z 747.937,A -85,B 0,C 180,E1 -31326.555,E2 -31326.555} C_VEL
LIN {X 0,Y 34.657,Z 760.262,A -85,B 0,C 180,E1 -31328.588,E2 -31328.588} C_VEL
LIN {X 0,Y 27.911,Z 772.962,A -85,B 0,C 180,E1 -31332.581,E2 -31332.581} C_VEL
LIN {X 0,Y 20.777,Z 783.857,A -85,B 0,C 180,E1 -31339.774,E2 -31339.774} C_VEL
LIN {X 0,Y 14.619,Z 792.32,A -85,B 0,C 180,E1 -31352.831,E2 -31352.831} C_VEL
LIN {X 0,Y 9.549,Z 800.733,A -85,B 0,C 180,E1 -31388.36,E2 -31388.36} C_VEL
LIN {X 0,Y 10.999,Z 807.703,A -85,B 0,C 180,E1 -31438.59,E2 -31438.59} C_VEL
LIN {X 0,Y 13.576,Z 810.656,A -85,B 0,C 180,E1 -31457.987,E2 -31457.987} C_VEL
LIN {X 0,Y 14.914,Z 811.76,A -85,B 0,C 180,E1 -31471.88,E2 -31471.88} C_VEL
LIN {X 0,Y 7.494,Z 803.59,A -85,B 0,C 180,E1 -31520.487,E2 -31520.487} C_VEL
LIN {X 0,Y 10.625,Z 794.892,A -85,B 0,C 180,E1 -31582.885,E2 -31582.885} C_VEL
LIN {X 0,Y 18.117,Z 784.92,A -85,B 0,C 180,E1 -31604.126,E2 -31604.126} C_VEL
LIN {X 0,Y 25.55,Z 774.193,A -85,B 0,C 180,E1 -31611.828,E2 -31611.828} C_VEL
LIN {X 0,Y 32.205,Z 762.605,A -85,B 0,C 180,E1 -31615.893,E2 -31615.893} C_VEL
LIN {X 0,Y 37.367,Z 751.499,A -85,B 0,C 180,E1 -31617.98,E2 -31617.98} C_VEL
LIN {X 0,Y 41.851,Z 738.72,A -85,B 0,C 180,E1 -31619.493,E2 -31619.493} C_VEL
LIN {X 0,Y 45.215,Z 724.803,A -85,B 0,C 180,E1 -31620.553,E2 -31620.553} C_VEL
LIN {X 0,Y 49.175,Z 702.608,A -85,B 0,C 180,E1 -31621.774,E2 -31621.774} C_VEL
LIN {X 0,Y 49.127,Z 700.444,A -85,B 0,C 180,E1 -31622.879,E2 -31622.879} C_VEL
LIN {X 0,Y 48.241,Z 694.17,A -85,B 0,C 180,E1 -31628.538,E2 -31628.538} C_VEL
LIN {X 0,Y 47.268,Z 690.337,A -85,B 0,C 180,E1 -31634.307,E2 -31634.307} C_VEL
LIN {X 0,Y 46.525,Z 687.546,A -85,B 0,C 180,E1 -31640.782,E2 -31640.782} C_VEL
LIN {X 0,Y 46.255,Z 685.797,A -85,B 0,C 180,E1 -31646.476,E2 -31646.476} C_VEL
LIN {X 0,Y 46.088,Z 685.706,A -85,B 0,C 180,E1 -31651.222,E2 -31651.222} C_VEL
LIN {X 0,Y 45.969,Z 686.443,A -85,B 0,C 180,E1 -31653.762,E2 -31653.762} C_VEL
LIN {X 0,Y 45.664,Z 688.644,A -85,B 0,C 180,E1 -31656.223,E2 -31656.223} C_VEL
LIN {X 0,Y 45.128,Z 693.472,A -85,B 0,C 180,E1 -31660.42,E2 -31660.42} C_VEL
LIN {X 0,Y 45.5,Z 699.167,A -85,B 0,C 180,E1 -31668.774,E2 -31668.774} C_VEL
LIN {X 0,Y 45.668,Z 702.487,A -85,B 0,C 180,E1 -31671.87,E2 -31671.87} C_VEL
LIN {X 0,Y 45.632,Z 708.057,A -85,B 0,C 180,E1 -31675.455,E2 -31675.455} C_VEL
LIN {X 0,Y 40.897,Z 733.052,A -85,B 0,C 180,E1 -31676.402,E2 -31676.402} C_VEL
LIN {X 0,Y 36.954,Z 746.4,A -85,B 0,C 180,E1 -31677.043,E2 -31677.043} C_VEL
LIN {X 0,Y 32.54,Z 757.138,A -85,B 0,C 180,E1 -31677.617,E2 -31677.617} C_VEL
LIN {X 0,Y 26.37,Z 768.815,A -85,B 0,C 180,E1 -31678.628,E2 -31678.628} C_VEL
LIN {X 0,Y 18.887,Z 780.065,A -85,B 0,C 180,E1 -31680.867,E2 -31680.867} C_VEL
LIN {X 0,Y 10.631,Z 790.25,A -85,B 0,C 180,E1 -31687.096,E2 -31687.096} C_VEL
LIN {X 0,Y 2.852,Z 798.968,A -85,B 0,C 180,E1 -31731.771,E2 -31731.771} C_VEL
LIN {X 0,Y 2.409,Z 800.484,A -85,B 0,C 180,E1 -31769.819,E2 -31769.819} C_VEL
LIN {X 0,Y 1.837,Z 801.039,A -85,B 0,C 180,E1 -31819.015,E2 -31819.015} C_VEL
LIN {X 0,Y 6.193,Z 793.694,A -85,B 0,C 180,E1 -31981.715,E2 -31981.715} C_VEL
LIN {X 0,Y 14.352,Z 784.468,A -85,B 0,C 180,E1 -31985.774,E2 -31985.774} C_VEL
LIN {X 0,Y 22.271,Z 773.66,A -85,B 0,C 180,E1 -31987.014,E2 -31987.014} C_VEL
LIN {X 0,Y 28.918,Z 762.449,A -85,B 0,C 180,E1 -31987.832,E2 -31987.832} C_VEL
LIN {X 0,Y 34.367,Z 750.94,A -85,B 0,C 180,E1 -31988.211,E2 -31988.211} C_VEL
LIN {X 0,Y 39.265,Z 736.977,A -85,B 0,C 180,E1 -31988.621,E2 -31988.621} C_VEL
LIN {X 0,Y 42.45,Z 723.45,A -85,B 0,C 180,E1 -31988.995,E2 -31988.995} C_VEL
LIN {X 0,Y 46.058,Z 703.515,A -85,B 0,C 180,E1 -31989.714,E2 -31989.714} C_VEL
LIN {X 0,Y 45.653,Z 698.615,A -85,B 0,C 180,E1 -31994.614,E2 -31994.614} C_VEL
LIN {X 0,Y 45.091,Z 694.962,A -85,B 0,C 180,E1 -32001.433,E2 -32001.433} C_VEL
LIN {X 0,Y 44.925,Z 692.749,A -85,B 0,C 180,E1 -32008.205,E2 -32008.205} C_VEL
LIN {X 0,Y 45.123,Z 692.964,A -85,B 0,C 180,E1 -32019.478,E2 -32019.478} C_VEL
LIN {X 0,Y 45.128,Z 693.472,A -85,B 0,C 180,E1 -32020.42,E2 -32020.42} C_VEL
LIN {X 0,Y 44.959,Z 696.628,A -85,B 0,C 180,E1 -32023.5,E2 -32023.5} C_VEL
LIN {X 0,Y 44.449,Z 701.631,A -85,B 0,C 180,E1 -32025.904,E2 -32025.904} C_VEL
LIN {X 0,Y 43.388,Z 708.471,A -85,B 0,C 180,E1 -32026.95,E2 -32026.95} C_VEL
LIN {X 0,Y 42.346,Z 714.013,A -85,B 0,C 180,E1 -32026.847,E2 -32026.847} C_VEL
LIN {X 0,Y 38.243,Z 734.385,A -85,B 0,C 180,E1 -32026.691,E2 -32026.691} C_VEL
LIN {X 0,Y 34.385,Z 746.85,A -85,B 0,C 180,E1 -32026.182,E2 -32026.182} C_VEL
LIN {X 0,Y 29.126,Z 759.135,A -85,B 0,C 180,E1 -32024.892,E2 -32024.892} C_VEL
LIN {X 0,Y 23.287,Z 769.855,A -85,B 0,C 180,E1 -32022.887,E2 -32022.887} C_VEL
LIN {X 0,Y 15.248,Z 781.78,A -85,B 0,C 180,E1 -32017.264,E2 -32017.264} C_VEL
LIN {X 0,Y 15.141,Z 781.796,A -85,B 0,C 180,E1 -32012.348,E2 -32012.348} C_VEL
LIN {X 0,Y 22.637,Z 770.396,A -85,B 0,C 180,E1 -32004.406,E2 -32004.406} C_VEL
LIN {X 0,Y 29.211,Z 758.102,A -85,B 0,C 180,E1 -32001.155,E2 -32001.155} C_VEL
LIN {X 0,Y 34.344,Z 745.804,A -85,B 0,C 180,E1 -31999.539,E2 -31999.539} C_VEL
LIN {X 0,Y 38.342,Z 732.705,A -85,B 0,C 180,E1 -31998.636,E2 -31998.636} C_VEL
LIN {X 0,Y 43.301,Z 707.532,A -85,B 0,C 180,E1 -31998.129,E2 -31998.129} C_VEL
LIN {X 0,Y 43.621,Z 705.434,A -85,B 0,C 180,E1 -31998.505,E2 -31998.505} C_VEL
LIN {X 0,Y 43.617,Z 703.058,A -85,B 0,C 180,E1 -32001.491,E2 -32001.491} C_VEL
LIN {X 0,Y 43.587,Z 700.332,A -85,B 0,C 180,E1 -32007.73,E2 -32007.73} C_VEL
LIN {X 0,Y 43.6,Z 699.692,A -85,B 0,C 180,E1 -32011.082,E2 -32011.082} C_VEL
LIN {X 0,Y 43.659,Z 699.816,A -85,B 0,C 180,E1 -32016.277,E2 -32016.277} C_VEL
LIN {X 0,Y 43.478,Z 704.207,A -85,B 0,C 180,E1 -32022.791,E2 -32022.791} C_VEL
LIN {X 0,Y 43.214,Z 708.915,A -85,B 0,C 180,E1 -32026.465,E2 -32026.465} C_VEL
LIN {X 0,Y 42.462,Z 713.419,A -85,B 0,C 180,E1 -32026.883,E2 -32026.883} C_VEL
LIN {X 0,Y 42.346,Z 714.013,A -85,B 0,C 180,E1 -32026.847,E2 -32026.847} C_VEL
LIN {X 0,Y 41.094,Z 719.747,A -85,B 0,C 180,E1 -32025.655,E2 -32025.655} C_VEL
LIN {X 0,Y 36.751,Z 736.145,A -85,B 0,C 180,E1 -32017.239,E2 -32017.239} C_VEL
LIN {X 0,Y 34.779,Z 742.61,A -85,B 0,C 180,E1 -32014.965,E2 -32014.965} C_VEL
LIN {X 0,Y 34.466,Z 743.544,A -85,B 0,C 180,E1 -32014.843,E2 -32014.843} C_VEL
LIN {X 0,Y 31.569,Z 751.604,A -85,B 0,C 180,E1 -32012.966,E2 -32012.966} C_VEL
LIN {X 0,Y 36.092,Z 738.072,A -85,B 0,C 180,E1 -32010.089,E2 -32010.089} C_VEL
LIN {X 0,Y 39.222,Z 724.569,A -85,B 0,C 180,E1 -32008.589,E2 -32008.589} C_VEL
LIN {X 0,Y 42.167,Z 708.244,A -85,B 0,C 180,E1 -32007.842,E2 -32007.842} C_VEL
LIN {X 0,Y 42.339,Z 706.697,A -85,B 0,C 180,E1 -32011.65,E2 -32011.65} C_VEL
LIN {X 0,Y 42.301,Z 706.898,A -85,B 0,C 180,E1 -32013.117,E2 -32013.117} C_VEL
LIN {X 0,Y 41.96,Z 709.286,A -85,B 0,C 180,E1 -32016.234,E2 -32016.234} C_VEL
LIN {X 0,Y 41.738,Z 710.879,A -85,B 0,C 180,E1 -32017.379,E2 -32017.379} C_VEL
LIN {X 0,Y 37.313,Z 733.597,A -85,B 0,C 180,E1 -32016.061,E2 -32016.061} C_VEL
LIN {X 0,Y 34.466,Z 743.544,A -85,B 0,C 180,E1 -32014.843,E2 -32014.843} C_VEL
LIN {X 0,Y 34.466,Z 743.544,A -85,B 0,C 180,E1 -32014.843,E2 -32014.843}

QRS_NEXT_CUT()

QRS_NEXT()
QRS_HOME()

END
